(* PLC project BasePpt, Beckhoff Automation GmbH TwinCAT PLC Control 3.5.6.0 *)
(* stored: creationDateTime 2015-05-28T16:00:50.6422414, modificationDateTime 2015-05-28T16:00:50.6452414 *)

TYPE T_Ctrl_SIf_IBH : STRUCT
  Cfg : T_Ctrl_SIf_IBH_Cfg;  (* configuration *)
  Par : T_Ctrl_SIf_IBH_Par;  (* parameter *)
  Cur : T_Ctrl_SIf_IBH_Cur;  (* current values *)
END_STRUCT;
END_TYPE

TYPE T_Ctrl_SIf_IBH_Cfg : STRUCT
  uiNumberOfModules : UINT;  (* Number of Modules in use, <= 8 *)
  tIpAddress : T_IPv4Addr;  (* IPv4 network address *)
  udiPortAdress : UDINT;  (* Remote (server) port address *)
  nDeviceAddress : BYTE;  (* MPI device address *)
  nDatablockNumber : BYTE;  (* Read/write from/to datablock number *)
  tTimeout : TIME;  (* Maximum time allowed for the execution of the command *)
  nWriteStartAddress : WORD;  (* Write byte/word offset/start address *)
  nReadStartAddress : WORD;  (* Read byte/word offset/start address *)
  uiByteOffset_rd_iStatus : UINT;
  uiByteOffset_rd_bOff : UINT;
  uiBitOffset_rd_bOff : UINT;
  uiByteOffset_rd_bBeltOn : UINT;
  uiBitOffset_rd_bBeltOn : UINT;
  uiByteOffset_rd_bManual : UINT;
  uiBitOffset_rd_bManual : UINT;
  uiByteOffset_rd_bRun : UINT;
  uiBitOffset_rd_bRun : UINT;
  uiByteOffset_rd_bSetParam : UINT;
  uiBitOffset_rd_bSetParam : UINT;
  uiByteOffset_rd_bGetParam : UINT;
  uiBitOffset_rd_bGetParam : UINT;
  uiByteOffset_rd_bAckError : UINT;
  uiBitOffset_rd_bAckError : UINT;
  uiByteOffset_rd_adiTemp_mc : UINT;
  uiByteOffset_rd_adiAir_p : UINT;
  uiByteOffset_rd_diSpeed_mm_min : UINT;
  uiByteOffset_rd_iErrorLevel : UINT;
  uiByteOffset_rd_iErrorID : UINT;
  uiByteOffset_rd_iErrorValue : UINT;
  uiByteOffset_wr_iOff : UINT;
  uiByteOffset_wr_iBeltOn : UINT;
  uiByteOffset_wr_iManual : UINT;
  uiByteOffset_wr_iRun : UINT;
  uiByteOffset_wr_iSetParam : UINT;
  uiByteOffset_wr_iGetParam : UINT;
  uiByteOffset_wr_iAckError : UINT;
  uiByteOffset_wr_adiTemp_mc : UINT;
  uiByteOffset_wr_adiAir_p : UINT;
  uiByteOffset_wr_diSpeed_mm_min : UINT;
END_STRUCT;
END_TYPE

TYPE T_Ctrl_SIf_IBH_Cur : STRUCT

END_STRUCT;
END_TYPE

TYPE T_Ctrl_SIf_IBH_Par : STRUCT

END_STRUCT;
END_TYPE

TYPE E_AmpType : (BOTH_ROT_LIN := 0, ROTARY_AMP := 1, LINEAR_AMP := 2) USINT;
END_TYPE

(* values of E_POD_UseHomeSwitch: SI0: internal IO 2 Home switch 0: Switched off, 1: Switched on; SI1: internal IO 16 SI0: 0: Switched off (Open),1: Switched on (Close); SI2: internal IO 17 SI0: 0: Switched off (Open),1: Switched on (Close); SI3: internal IO 18 SI0: 0: Switched off (Open),1: Switched on (Close); SI4: internal IO 19 SI0: 0: Switched off (Open),1: Switched on (Close); SI5: internal IO 20 SI0: 0: Switched off (Open),1: Switched on (Close); SI6: internal IO 21 SI0: 0: Switched off (Open),1: Switched on (Close) internal IO 22 SI0: 0: Switched off (Open),1: Switched on (Close) *)

TYPE E_POD_UseHomeSwitch : (FUB_Input := 0, HomeSwitch, SI0, SI1, SI2, SI3, SI4, SI5, SI6) USINT;
END_TYPE

TYPE E_ValueType : (TYPE_NOT_SPECIFIED := 0, TYPE_SINT := 1, TYPE_INT := 2, TYPE_DINT := 3, TYPE_USINT := 4, TYPE_UINT := 5, TYPE_UDINT := 6, TYPE_STRING := 7) USINT;
END_TYPE

TYPE T_POD : STRUCT
  strAxisName : STRING(31);
  strState : STRING;
  strCmd : STRING;
  intCmd : INT;
  intServiceCmd : INT;
  stStatus : T_POD_Status;
  stMove : T_POD_Move;
  stErr : T_POD_Error;
  stCfg : T_POD_Cfg;
  stService : T_POD_Service;
END_STRUCT;
END_TYPE

TYPE T_POD_Cfg : STRUCT
  bolSimulation : BOOL;
  lreHomePosition : LREAL;  (* >0 Homeposition set if calibsignal active *)
  eHomingMode : MC_HomingMode;  (* Home Mode *)
  eUseHomeSwitch : E_POD_UseHomeSwitch;  (* define home switch: 0 use FUB input, *)
END_STRUCT;
END_TYPE

TYPE T_POD_DigitalInputs : STRUCT
  bol_N_OT : BOOL;  (* 0 N-OT: Negative limit switch 0: Switched off, 1: Switched on *)
  bol_P_OT : BOOL;  (* 1 P-OT: Positive limit switch 0: Switched off, 1: Switched on *)
  bol_HomeSwitch : BOOL;  (* 2 Home switch 0: Switched off, 1: Switched on *)
  bol_SI0 : BOOL;  (* 16 SI0: CN1-13pin 0: Switched off (Open),1: Switched on (Close) *)
  bol_SI1 : BOOL;  (* 17 SI1: CN1-7pin 0: Switched off (Open),1: Switched on (Close) *)
  bol_SI2 : BOOL;  (* 18 SI2: CN1-8pin 0: Switched off (Open),1: Switched on (Close) *)
  bol_SI3 : BOOL;  (* 19 SI3: CN1-9pin 0: Switched off (Open),1: Switched on (Close) *)
  bol_SI4 : BOOL;  (* 20 SI4: CN1-10pin 0: Switched off (Open),1: Switched on (Close) *)
  bol_SI5 : BOOL;  (* 21 SI5: CN1-11pin 0: Switched off (Open),1: Switched on (Close) *)
  bol_SI6 : BOOL;  (* 22 SI6: CN1-12pin 0: Switched off (Open),1: Switched on (Close) *)
END_STRUCT;
END_TYPE

TYPE T_POD_Error : STRUCT
  bolErrAck : BOOL;  (* Reset failure *)
  bolErrorActive : BOOL;  (* atleast one failure active *)
  bolMCError : BOOL;  (* error in MC fub error *)
  bolNCError : BOOL;  (* error in NC (motion controller) *)
  bolDriveError : BOOL;  (* error in drive (ELMO) *)
  dwoErrorID : DWORD;  (* error ID *)
END_STRUCT;
END_TYPE

TYPE T_POD_Move : STRUCT
  lreSetPos : LREAL;  (* target position [Units] *)
  eDirection : MC_Direction;  (* Direction used for Modulo position *)
  lreSetSpeed : LREAL;  (* set speed [Units/s] *)
  lreSetAcc : LREAL;  (* set acc [Units/s^2] *)
  lreSetDec : LREAL;  (* set dec [Units/s^2] *)
  lreSetDecFast : LREAL;  (* set dec [Units/s^2] quickstop *)
  lreSetJerk : LREAL;  (* lreSetDec : DINT; //set dec [Units/s^2] *)
  lreSpeedOverride : LREAL := 100.0;  (* speed override for all drive commands (0 ≤Override≤ 100.0) *)
  lreSWLimitNeg_mm : LREAL;
  lreSWLimitPos_mm : LREAL;
  lreActPos : LREAL;  (* Actual position [Units] *)
  lreActModPos : LREAL;  (* Actual modulo position [Units] *)
  lreActVel : LREAL;  (* act speed [Units/s] *)
  lreActTorque : LREAL;  (* [Nm] actual torque The torque actual value corresponds to the instantaneous torque in the drive motor. The value is given in units of per thousand of rated torque. *)
END_STRUCT;
END_TYPE

TYPE T_POD_Service : STRUCT
  worIndex : WORD;  (* Index of the object that should be written to. *)
  bytSubIndex : BYTE;  (* Sub-index of the object that should be written to. *)
  dwo_pSrcBuf : DWORD;  (* Address (pointer) of the send buffer. *)
  udi_cbBufLen : UDINT;  (* Number (in bytes) of data to be sent. *)
  eValueType : E_ValueType;  (* value type *)
  eNC_ParNumber : MC_AxisParameter;  (* parameter number of read/write NC parameters *)
  strValue : STRING;  (* write/read value if dwo_pSrcBuf = 0 *)
END_STRUCT;
END_TYPE

TYPE T_POD_StateMachine : STRUCT
  intState : INT;  (* actual state *)
  intStateLastCycle : INT;  (* state of last cycle *)
  intStateHistory : INT;  (* save history backup p.e. in ERROR state *)
  intStateNext : INT;  (* set state for next cycle *)
END_STRUCT;
END_TYPE

TYPE T_POD_Status : STRUCT
  bolEnable : BOOL;  (* Hardware enable:0 = Open 1 = Closed *)
  bolNetwOk : BOOL;  (* 1 = Network initialized *)
  bolInitOk : BOOL;  (* 1 = Initialization done *)
  bolReady : BOOL;
  bolCtrlOn : BOOL;  (* 1 = Controller switched on *)
  bolHomeOk : BOOL;  (* 1 = Homing done *)
  bolInPos : BOOL;  (* 1 = In position (target position reached) *)
  bolMoving : BOOL;  (* 1 = Axis moving *)
  bolNegHWSwitch : BOOL;  (* 1 = negativ endswitch active -> no movement negative allowed *)
  bolPosHWSwitch : BOOL;  (* 1 = positive endswitch active -> no movement positive allowed *)
  bolNegSWSwitch : BOOL;  (* 1 = negativ endswitch active -> no movement negative allowed *)
  bolPosSWSwitch : BOOL;  (* 1 = positive endswitch active -> no movement positive allowed *)
  stDigIn : T_POD_DigitalInputs;  (* drive digital inputs of elmo drive *)
END_STRUCT;
END_TYPE

TYPE T_POD_StatusWord : STRUCT
  bolReadyToSwitchOn : BOOL;  (* 0 Ready TO Switch on =1 *)
  bolSwitchedOn : BOOL;  (* 1 Switched on =1 *)
  bolOperationEnabled : BOOL;  (* 2 Operation enabeld =1 *)
  bolFault : BOOL;  (* 3 Fault/Fault Reaction *)
  bolMainPowerOn : BOOL;  (* 4 MainPower on =1 *)
  bolQuickStopInactive : BOOL;  (* 5 Quickstop inaktive =1 *)
  bolSwitchOnDisabled : BOOL;  (* 6 Switch on disabled =1 *)
  bolWarning : BOOL;  (* 7 Warning is occurred =1 *)
  bolBit08 : BOOL;  (* 8 not used always 0 *)
  bolRemote : BOOL;  (* 9 The Remote bit is always set by the Elmo servo drive *)
  bolTargetReached : BOOL;  (* 10 Target Reached *)
  bolInternLimit : BOOL;  (* 11 Internal Limit active =1 *)
END_STRUCT;
END_TYPE

TYPE E_PTR_Status : (EnterBusy, OnBelt, ExitBusy, Gone, ERROR, MAX_E_PTR_Status);
END_TYPE

TYPE T_PTR_STRUCT : STRUCT
  udiTimeOnBelt_us : UDINT;  (* [us] Time of the paper on the belt *)
  lrePositionOnBelt_mm : LREAL;  (* [mm] Position of the paper on the belt *)
  lrePositionOnBeltAdjusted_mm : LREAL;  (* [mm] Position of the paper on the belt Adjusted to the possible maximum *)
  udiItemId : UDINT;  (* Paper Item Id *)
  eStatus : E_PTR_Status;  (* Error *)
END_STRUCT;
END_TYPE

TYPE E_ALM_TCP : (SocketConnectionLost := 1, AddToSendBufferFailed := 2, RemoveFromSendBufferFailed := 3, GetFromSendBufferFailed := 4, AddToReceiveBufferFailed := 5, RemoveFromReceiveBufferFailed := 6, GetFromReceiveBufferFailed := 7, NotSent := 8, NoAckReceived := 9, FubErrorClientConnection := 10, FubErrorSendData := 11, FubErrorReceiveData := 12, MAX_E_ALM_TCP) UINT;
END_TYPE

{attribute 'pack_mode' := '1'}
TYPE ST_Header : STRUCT
  uinMsgId : UINT;
  udiMsgSize : UDINT;
END_STRUCT;
END_TYPE

TYPE T_Ctrl_SIf_TCP : STRUCT
  Cfg : T_Ctrl_SIf_TCP_Cfg;  (* configuration *)
  Par : T_Ctrl_SIf_TCP_Par;  (* parameter *)
  Cur : T_Ctrl_SIf_TCP_Cur;  (* current values *)
  Alm : ARRAY[1..(E_ALM_TCP.MAX_E_ALM_TCP - 1)] OF T_Ctrl_Alm;  (* alarm number used in this controller *)
END_STRUCT;
END_TYPE

TYPE T_Ctrl_SIf_TCP_Cfg : STRUCT
  bUsingAck : BOOL;  (* depending on the protocol an ACK is used or not *)
  bolAutoReconnectEnable : BOOL;  (* Enable Auto Reconnect *)
END_STRUCT;
END_TYPE

TYPE T_Ctrl_SIf_TCP_Cur : STRUCT
  bolFubErrorActive : BOOL;
END_STRUCT;
END_TYPE

TYPE T_Ctrl_SIf_TCP_Par : STRUCT
  strIPAdr : STRING(15);
  udiPort : UDINT;
  tTOConnection : TIME;
  tTOReceive : TIME;
  tTOSend : TIME;
  iMaxWaitTimeAck : TIME;
  iMaxSendTry : USINT;
END_STRUCT;
END_TYPE

TYPE E_ALM_GRR : (NONE := 1, SystemError := 2, MainPressureError := 3, EoffOrFuseError := 4, LowPowderWarning := 5, ManualOperation := 6, LostConnection := 7, MAX_E_ALM_GRR) UINT;
END_TYPE

TYPE T_Ctrl_SIf_GRR : STRUCT
  Cfg : T_Ctrl_SIf_GRR_Cfg;  (* configuration *)
  Par : T_Ctrl_SIf_GRR_Par;  (* parameter *)
  Cur : T_Ctrl_SIf_GRR_Cur;  (* current values *)
  In : T_Ctrl_SIf_GRR_In;  (* io input *)
  Out : T_Ctrl_SIf_GRR_Out;  (* io output *)
  Alm : ARRAY[1..(E_ALM_GRR.MAX_E_ALM_GRR - 1)] OF T_Ctrl_Alm;  (* alarm number used in this controller *)
END_STRUCT;
END_TYPE

TYPE T_Ctrl_SIf_GRR_Cfg : STRUCT
  rMaxFreq_Hz : REAL;
END_STRUCT;
END_TYPE

TYPE T_Ctrl_SIf_GRR_Cur : STRUCT
  intMainPressure : INT;
END_STRUCT;
END_TYPE

TYPE T_Ctrl_SIf_GRR_In : STRUCT
  bolSystemOk : T_Ctrl_IoBool;
  bolMainPressureError : T_Ctrl_IoBool;
  bolEoffOrFuseOk : T_Ctrl_IoBool;
  bolPowderLowWarning : T_Ctrl_IoBool;
  bolAutoMode : T_Ctrl_IoBool;
  intState : T_Ctrl_IoInt;
  bolToggleBitGrn : T_Ctrl_IoBool;
  intMainPressure : T_Ctrl_IoInt;
END_STRUCT;
END_TYPE

TYPE T_Ctrl_SIf_GRR_Out : STRUCT
  intCommand : BASE_PLC.T_Ctrl_IoInt;
  intConveyorBelt : T_Ctrl_IoInt;
  intPowderVibrator : T_Ctrl_IoInt;
  intConveyorVibrator : T_Ctrl_IoInt;
  intAnalogValue : T_Ctrl_IoInt;
  uinFilterClearingCycleTime_min : T_Ctrl_IoUint;
  bolToggleBitGrr : T_Ctrl_IoBool;
END_STRUCT;
END_TYPE

TYPE T_Ctrl_SIf_GRR_Par : STRUCT
  rConveyorBelt_Hz : REAL;
  rPowderVibrator_Hz : REAL;
  rConveyorVibrator_Hz : REAL;
  rAnalogValue_p : REAL;
  uinFilterClearingCycleTime_min : UINT;
END_STRUCT;
END_TYPE

TYPE E_ALM_JCL : (NONE := 1, JetterNotRun := 2, JetterManualWarning := 3, JetterManualError := 4, JetterEOff := 5, JetterCommunicationLost := 6, CleaningError, MAX_E_ALM_JCL) UINT;
END_TYPE

TYPE T_Ctrl_SIf_JCL : STRUCT
  Cfg : T_Ctrl_SIf_JCL_Cfg;  (* configuration *)
  Par : T_Ctrl_SIf_JCL_Par;  (* parameter *)
  Cur : T_Ctrl_SIf_JCL_Cur;  (* current values *)
  Alm : ARRAY[1..(E_ALM_JCL.MAX_E_ALM_JCL - 1)] OF T_Ctrl_Alm;  (* alarm number used in this controller *)
END_STRUCT;
END_TYPE

TYPE T_Ctrl_SIf_JCL_Cfg : STRUCT
  bolJetterManualModeAllowed : BOOL;  (* FALSE = Do not allow manual mode, go to error if Jetter goes to manual / TRUE = Allow manual mode and stay in the last state *)
END_STRUCT;
END_TYPE

TYPE T_Ctrl_SIf_JCL_Cur : STRUCT
  bolIsLocalControlled : BOOL;  (* Additional states from TCP server Local control active. Commands from this client are ignored *)
  bolIsRemoteControlled : BOOL;  (* Remote control active. Commands from this client are accepted *)
  bolReadyForProduction : BOOL;  (* Jetter ready for production *)
  bolMaintenanceInProgress : BOOL;  (* TRUE if a maintenance work is in progress. Independent if auto or manual maintenance is in progress. *)
  bolRunning : BOOL;  (* Print running, in production *)
  bolNeedsAttention : BOOL;  (* System needs attention. Info or warning active *)
  bolError : BOOL;  (* General error active *)
  bolCleaningIncomplete : BOOL;  (* Cleaning cycle was aborted before finishing. Production not possible. *)
  bolNeedsCleaning : BOOL;  (* Print head needs cleaning. *)
  strDTOfLastCleaningCycle : STRING := '';  (* Timestamp of the last cleaning cycle. Format: YYYY-MM-DD-hh:mm:ss.xxx *)
  intJETState : INT;  (* Jetter state *)
END_STRUCT;
END_TYPE

TYPE T_Ctrl_SIf_JCL_Par : STRUCT
  udiCleaningStartTimeout_ms : UDINT;  (* [ms] Timeout to detect cleaning start failure *)
END_STRUCT;
END_TYPE

TYPE T_JCL_AlmMsg : STRUCT
  stHeader : ST_Header;
  udiAlarmID : UDINT;  (* Unique alarm number *)
  udiInfo : UDINT;  (* Additional information *)
  usiClass : USINT;  (* Corresponding alarm class *)
  uinCtrlID : UINT;  (* Corresponding controller ID *)
  strDTEntry : STRING(25);  (* Entry date and time *)
  strText : STRING(255);  (* Alarm Text *)
END_STRUCT;
END_TYPE

{attribute 'pack_mode' := '1'}
TYPE T_JCL_Command : STRUCT
  stHeader : ST_Header;
  usiCommand : USINT;
END_STRUCT;
END_TYPE

TYPE T_JCL_PrintDone : STRUCT
  stHeader : ST_Header;
  usiBarcode : ARRAY[0..9] OF USINT;
  usiInkLevelMainTank : USINT;  (* [%] *)
  usiInkLevelSupplyPrintModule1 : USINT;  (* [%] *)
  usiInkLevelSupplyPrintModule2 : USINT;  (* [%] *)
  usiInkLevelReturnPrintModule1 : USINT;  (* [%] *)
  usiInkLevelReturnPrintModule2 : USINT;  (* [%] *)
  udiInkMeniscus : ARRAY[0..1] OF UDINT;  (* [0.01 mbar] *)
  udiPrintHeadTemperature : ARRAY[0..1, 0..4] OF UDINT;  (* [0.1 °C] *)
  udiPrintWidthCalc : UDINT;  (* [Micrometer] // Dimension of printed file calculated by DJM *)
  udiPrintLengthCalc : UDINT;  (* [Micrometer] // Dimension of printed file calculated by DJM *)
  udiShiftXCalc : UDINT;  (* [Micrometer] // Offset of print *)
  udiShiftYCalc : UDINT;  (* [Micrometer] // Offset of print *)
  udiShiftAngleCalc : UDINT;  (* [0.01°] // Offset of rotation angle *)
END_STRUCT;
END_TYPE

{attribute 'pack_mode' := '1'}
TYPE T_JCL_RequestCleaning : STRUCT
  stHeader : ST_Header;
  strDTLastClean : STRING(25);  (* Date and time of the last cleaning cycle *)
  uinRequiredInterval_min : UINT;  (* Required interval for cleaning [min] *)
END_STRUCT;
END_TYPE

{attribute 'pack_mode' := '1'}
TYPE T_JCL_State : STRUCT
  stHeader : ST_Header;
  usiMainState : USINT;
  usiAddState : USINT;  (* (Bit coded) *)
END_STRUCT;
END_TYPE

{attribute 'qualified_only'}
TYPE E_ALM_RAX : (GeneralDrive := 1, GeneralNc, SwLimit, NegHwLimit, PosHwLimit, InterlockNegMove, InterlockPosMove, GeneralMCFUB, MAX_E_ALM) UINT;
END_TYPE

TYPE T_Ctrl_SIf_RAX : STRUCT
  Cfg : T_Ctrl_SIf_RAX_Cfg;  (* configuration *)
  Par : T_Ctrl_SIf_RAX_Par;  (* parameter *)
  Cur : T_Ctrl_SIf_RAX_Cur;  (* current values *)
  Alm : ARRAY[1..(E_ALM_RAX.MAX_E_ALM - 1)] OF T_Ctrl_Alm;  (* alarm number used in this controller *)
  Ilk : T_Ctrl_SIf_RAX_Ilk;  (* interlock of output/movements *)
END_STRUCT;
END_TYPE

TYPE T_Ctrl_SIf_RAX_Cfg : STRUCT
  eHomingMode : MC_HomingMode;  (* homing mode *)
  lreShortestWayWindow_deg : LREAL;
END_STRUCT;
END_TYPE

TYPE T_Ctrl_SIf_RAX_Cur : STRUCT
  dinSpeed_0_1deg_s : DINT;  (* [0.1°/s] current speed *)
  dinPosition_0_1deg : DINT;  (* [0.1°] current position *)
  dinModPosition_0_1deg : DINT;  (* [°] current modulo position *)
  dinTorque_0_1Nm : DINT;  (* [0.1Nm] current torque *)
  bol_di1 : BOOL;  (* digital input1 from drive *)
  bol_di2 : BOOL;  (* digital input2 from drive *)
  bol_di3 : BOOL;  (* digital input3 from drive *)
  bol_di4 : BOOL;  (* digital input4 from drive *)
  bol_di5 : BOOL;  (* digital input5 from drive *)
END_STRUCT;
END_TYPE

TYPE T_Ctrl_SIf_RAX_Ilk : STRUCT
  bolMovePos : BOOL;  (* interlock movment in positive direction *)
  bolMoveNeg : BOOL;  (* interlock movment in negative direction *)
END_STRUCT;
END_TYPE

TYPE T_Ctrl_SIf_RAX_Par : STRUCT
  dinHomeOffset_0_1deg : DINT;  (* [deg] home offset *)
  dinPositionInit_0_1deg : DINT;  (* [0.1°] position init *)
  dinPos_0_1deg : DINT;  (* [0.1°] position absolute *)
  dinRelDist_0_1deg : DINT;  (* [0.1°] rel distance *)
  dinSpeed_0_1deg_s : DINT;  (* [0.1°/s] position speed *)
  dinSpeed_per : DINT;  (* [%] percent from dinSetSpeed_0_1deg_s *)
  dintAccDec_0_1deg_s2 : DINT;  (* [0.1°/s^2] position acceleration *)
  dinAcc_per : DINT;  (* [%] percent from dintAccDec_0_1deg_s2 *)
  dinDec_per : DINT;  (* [%] percent from dintAccDec_0_1deg_s2 *)
  dinSetDecFast_0_1deg_s2 : DINT;  (* [0.1°/s^2] position deceleration fast em stop *)
  dinSWLimitNeg_0_1deg : DINT;  (* [0.1°] negative sw limite *)
  dinSWLimitPos_0_1deg : DINT;  (* [0.1°] positive sw limite *)
END_STRUCT;
END_TYPE

TYPE E_ALM_BCH : (DataChannelMissing := 1, DataChannelBufferFull, BarcodeNotReadCorrectly, MAX_E_ALM_BCH) UINT;
END_TYPE

TYPE T_Ctrl_SIf_BCH : STRUCT
  Cfg : T_Ctrl_SIf_BCH_Cfg;  (* configuration *)
  Par : T_Ctrl_SIf_BCH_Par;  (* parameter *)
  Cur : T_Ctrl_SIf_BCH_Cur;  (* current values *)
  In : T_Ctrl_SIf_BCH_In;  (* Input layer *)
  Alm : ARRAY[1..(E_ALM_BCH.MAX_E_ALM_BCH - 1)] OF T_Ctrl_Alm;  (* alarm number used in this controller *)
END_STRUCT;
END_TYPE

TYPE T_Ctrl_SIf_BCH_Cfg : STRUCT
  bolEnableDataChannel : BOOL;  (* TRUE = Enable Data Channel; False = Disable DataChannel *)
  bolNegativeTriggerSignal : BOOL;  (* TRUE = Negative Trigger Signal, FALSE = Positive Trigger Signal *)
END_STRUCT;
END_TYPE

TYPE T_Ctrl_SIf_BCH_Cur : STRUCT

END_STRUCT;
END_TYPE

TYPE T_Ctrl_SIf_BCH_In : STRUCT
  bolSensorTrigScan : BASE_PLC.T_Ctrl_IoBool;  (* Trigger the measurement sensor *)
END_STRUCT;
END_TYPE

TYPE T_Ctrl_SIf_BCH_Par : STRUCT
  udiPaperGoneDelay_ms : UDINT;  (* [ms] Delay after the barcode has be read and the paper sensor signals that the paper is gone *)
  udiTestReadCylceTime_ms : UDINT;  (* [ms] Test Read Cycle Time *)
END_STRUCT;
END_TYPE

TYPE E_ALM_MDC : (TableSensorTimeout := 1, CrossSensorTimeout := 2, PositionSame := 3, MAX_E_ALM_MDC);
END_TYPE

TYPE T_Ctrl_SIf_MDC : STRUCT
  Cfg : T_Ctrl_SIf_MDC_Cfg;  (* configuration *)
  Par : T_Ctrl_SIf_MDC_Par;  (* parameter *)
  Cur : T_Ctrl_SIf_MDC_Cur;  (* current values *)
  In : T_Ctrl_SIf_MDC_In;  (* io input *)
  Out : T_Ctrl_SIf_MDC_Out;  (* io output *)
  Alm : ARRAY[1..MAX_E_ALM_MDC] OF T_Ctrl_Alm;  (* alarm number used in this controller *)
  Ilk : T_Ctrl_SIf_MDC_Ilk;  (* interlock of output/movements *)
END_STRUCT;
END_TYPE

TYPE T_Ctrl_SIf_MDC_Cfg : STRUCT
  uintPositionPerTurn : UINT;  (* Number of positions in 360° of the Malteser drive *)
END_STRUCT;
END_TYPE

TYPE T_Ctrl_SIf_MDC_Cur : STRUCT
  uintActualPosition : UINT;  (* Actual Position as position *)
  eActualTurningDirection : E_TURN_DIRECTION;  (* actual turning direction *)
  bolReferenceOk : BOOL;  (* Reference still ok *)
END_STRUCT;
END_TYPE

TYPE T_Ctrl_SIf_MDC_Ilk : STRUCT

END_STRUCT;
END_TYPE

TYPE T_Ctrl_SIf_MDC_In : STRUCT
  bolCrossPositionSensor : BASE_PLC.T_Ctrl_IoBool;  (* Is the cross in sensor positinon. One rotation step done. *)
  bolTablePositionSensor : BASE_PLC.T_Ctrl_IoBool;  (* Is the table at 0° degrees *)
END_STRUCT;
END_TYPE

TYPE T_Ctrl_SIf_MDC_Out : STRUCT
  intActualPosition : BASE_PLC.T_Ctrl_IoInt;
END_STRUCT;
END_TYPE

TYPE T_Ctrl_SIf_MDC_Par : STRUCT
  intTurnDirection : INT;  (* <0 = Turn left; =0 automatic; >0 turn right *)
  uinPositionToGo : UINT;  (* Position to go to if comand turn is given. 0 = initialization position *)
  udiStepRotationTime_ms : UDINT;  (* [ms] time to rotate one step *)
  udiInitializationTime_ms : UDINT;  (* [ms] initialization timeout time *)
  udiSimStepRotationTime_ms : UDINT;  (* [ms] simulation time to rotate one step *)
  udiSimInitializationTime_ms : UDINT;  (* [ms] simulation initialization timeout time *)
  udiSimStartRotationTime_ms : UDINT;  (* [ms] simulation time to start rotate and Cross sensor needs to go away *)
  uinPrePositionSpeed_rpm : UINT;  (* [rpm] PrePosition Speed *)
  uinPositionSpeed_rpm : UINT;  (* [rpm] Position Speed *)
END_STRUCT;
END_TYPE

(* values of E_ALM_OVN: Tesoma10000: OvertemperaturePowerSection - software reset - operating mode must be reelected; Tesoma10002: FailureOfActiveCoolingUnit; Tesoma10003: ActiveCoolingUnitNotRunning; Tesoma10006: FailureFuseGeneral - transport starts immediately when sensor is free; Tesoma10010: BeltPositionControlSensorError - software reset; Tesoma10011: BeltEdgeShutOff - software reset; Tesoma10012: FaultBeltSpeed - software reset; Tesoma10013: TransportOverload; Tesoma10014: BeltControlDeviceFault - software reset - reset FC; Tesoma10016: EmergencyStop - would be resettable, but since power is gone, the acknowledge does not arrive; Tesoma10023: BeltWearMonitor; Tesoma10024: ControlCabinetFan; Tesoma10025: ControlCabinetTemperatureTooHigh; Tesoma10026: PowerSupplyFailure; Tesoma10027: IntakeHoodTemperatureExceeded; Tesoma10030: AirPressureTooLow; Tesoma10031: BeltPositionControlNotWorking; Tesoma10032: ErrorCoolingDeviceControlCabinet; Tesoma10034: ControlCabinetCoolerAndSmallDrivesFuseFailure; Tesoma10x00: LimitSwitchingOff - software reset - after elimination, reactivates according zone; Tesoma10x01: OvertemperatureStl - software reset - after elimination AND reset, the STL reactivates the accordant zone; Tesoma10x02: FuseTriggered - software reset - after elimination, reactivates the accordant zone; Tesoma10x03: FailureExhaustAirDps - software reset - after elimination, reactivates the accordant zone; Tesoma10x07: ErrorFrequencyConverter - software reset - after elimination AND reset, the FC reactivates the accordant zone; Tesoma10x13: TemperatureSensorIrDefective; Tesoma10x14: FaultFrameCoolingSystemDps; Tesoma10x15: FaultExhaustAirDps; Tesoma13x00: TemperatureFault - software reset *)

TYPE E_ALM_OVN : (NONE := 0, TempError := 1, AirError := 2, SpeedError := 3, TimeoutError := 4, ParameterWarning := 5, ConnectionError := 6, WrongMode := 7, Tesoma10000 := 8, Tesoma10002 := 9, Tesoma10003 := 10, Tesoma10006 := 11, Tesoma10010 := 12, Tesoma10011 := 13, Tesoma10012 := 14, Tesoma10013 := 15, Tesoma10014 := 16, Tesoma10016 := 17, Tesoma10023 := 18, Tesoma10024 := 19, Tesoma10025 := 20, Tesoma10026 := 21, Tesoma10027 := 22, Tesoma10030 := 23, Tesoma10031 := 24, Tesoma10032 := 25, Tesoma10034 := 26, Tesoma10x00 := 27, Tesoma10x01 := 28, Tesoma10x02 := 29, Tesoma10x03 := 30, Tesoma10x07 := 31, Tesoma10x13 := 32, Tesoma10x14 := 33, Tesoma10x15 := 34, Tesoma13x00 := 35, TesomaUnknown := 36, HostConnectionLost := 37, SettingsChanged := 38, MAX_E_ALM_OVN);
END_TYPE

TYPE T_Ctrl_SIf_OVN : STRUCT
  Cfg : T_Ctrl_SIf_OVN_Cfg;  (* configuration *)
  Par : T_Ctrl_SIf_OVN_Par;  (* parameter *)
  Cur : T_Ctrl_SIf_OVN_Cur;  (* current values *)
  In : T_Ctrl_SIf_OVN_In;  (* io input *)
  Out : T_Ctrl_SIf_OVN_Out;  (* io output *)
  Alm : ARRAY[1..(E_ALM_OVN.MAX_E_ALM_OVN - 1)] OF T_Ctrl_Alm;  (* alarm number used in this controller *)
END_STRUCT;
END_TYPE

TYPE T_Ctrl_SIf_OVN_Cfg : STRUCT
  uiNumberOfModules : UINT;  (* Number of Modules in use *)
  diModuleLength_mm : DINT;  (* Length of one Module *)
  diDistanceBeforeOven_mm : DINT;  (* Distance before the first Module *)
  diDistanceAfterOven_mm : DINT;  (* Distance after the last Module *)
  diMaxSpeed_mm_min : DINT;  (* Maximal Belt Speed in mm/min *)
  diMinSpeed_mm_min : DINT;  (* Minimal Belt Speed in mm/min *)
  diMinTemp_dc : DINT;  (* Minimal Temperature in deci °C *)
  diMaxTemp_dc : DINT;  (* Maximal Temperature in deci °C *)
  diMinAir_p : DINT;  (* Minimal Airflow in % *)
  diMaxAir_p : DINT;  (* Maximal Airflow in % *)
  bAutoContinueAfterConnectionError : BOOL;  (* Auto Continue After Connection Error *)
  bolDataChannelEnable : BOOL;  (* Enable Data Channel *)
  bIgnoreOffBusyWaitPaper : BOOL;  (* ignore waiting for Paper to eject in OFFBusy *)
END_STRUCT;
END_TYPE

TYPE T_Ctrl_SIf_OVN_Cur : STRUCT
  diSpeed_mm_min : DINT;  (* Belt Speed in mm/min *)
  adiTemp_dc : ARRAY[0..(MAX_NUMBER_OF_OVEN_MODULES - 1)] OF DINT;  (* Temperature in deci °C *)
  adiAir_p : ARRAY[0..(MAX_NUMBER_OF_OVEN_MODULES - 1)] OF DINT;  (* Airflow in % *)
END_STRUCT;
END_TYPE

TYPE T_Ctrl_SIf_OVN_In : STRUCT

END_STRUCT;
END_TYPE

TYPE T_Ctrl_SIf_OVN_Out : STRUCT

END_STRUCT;
END_TYPE

TYPE T_Ctrl_SIf_OVN_Par : STRUCT
  diSpeed_mm_min : DINT;  (* Belt Speed in mm/min *)
  diSpeedBand1_mm_min : DINT;  (* Belt Speed Band in mm/min *)
  diSpeedBand2_mm_min : DINT;  (* Belt Speed Band in mm/min *)
  udiSpeedTimeout_ms : UDINT;  (* Belt Speed Timeout in ms *)
  adiTemp_dc : ARRAY[0..(MAX_NUMBER_OF_OVEN_MODULES - 1)] OF DINT;  (* Temperature in deci °C *)
  adiTempBand1_dc : ARRAY[0..(MAX_NUMBER_OF_OVEN_MODULES - 1)] OF DINT;  (* Temperature Band in deci °C *)
  adiTempBand2_dc : ARRAY[0..(MAX_NUMBER_OF_OVEN_MODULES - 1)] OF DINT;  (* Temperature Band in deci °C *)
  audiTempTimeout_ms : ARRAY[0..(MAX_NUMBER_OF_OVEN_MODULES - 1)] OF UDINT;  (* Temperature Timeout in ms *)
  adiAir_p : ARRAY[0..(MAX_NUMBER_OF_OVEN_MODULES - 1)] OF DINT;  (* Airflow in % *)
  adiAirBand1_p : ARRAY[0..(MAX_NUMBER_OF_OVEN_MODULES - 1)] OF DINT;  (* Airflow Band in % *)
  adiAirBand2_p : ARRAY[0..(MAX_NUMBER_OF_OVEN_MODULES - 1)] OF DINT;  (* Airflow Band in % *)
  audiAirTimeout_ms : ARRAY[0..(MAX_NUMBER_OF_OVEN_MODULES - 1)] OF UDINT;  (* Airflow Timeout in ms *)
  udiTimeoutOffBusy_ms : UDINT;
  udiTimeoutRunBusyReaction_ms : UDINT;
  udiTimeoutRunBusyInBand_ms : UDINT;
  udiTimeoutBeltOnlyReaction_ms : UDINT;
  udiTimeoutBeltOnlyBusy_ms : UDINT;
END_STRUCT;
END_TYPE

{attribute 'enable_dynamic_creation'}
TYPE T_Data : STRUCT
  uliBarcode : ULINT;
  bTrash : BOOL;
  diDistance_um : DINT;
  diSumTemp_mc : ARRAY[0..(MAX_NUMBER_OF_OVEN_MODULES - 1)] OF DINT;
  diCyclesInModule : ARRAY[0..(MAX_NUMBER_OF_OVEN_MODULES - 1)] OF DINT;
  bBarcodeMissed : BOOL;
END_STRUCT;
END_TYPE

TYPE E_ALM_PTB : (TestAlarm := 1, MAX_E_ALM_PTB);
END_TYPE

TYPE E_BELT_DIRECTION : (FORWARD := 0, BACKWARD := 1, MAX_E_BELT_DIRECTION);
END_TYPE

(* values of E_PTB_MODE: Endless: 0; ToSensor: 1; ToDistance: 2; ToTime: 3; Stack: 4 *)

TYPE E_PTB_MODE : (Endless, ToSensor, ToDistance, ToTime, Stack, MAX_E_PTB_MODE);
END_TYPE

TYPE E_PTB_PaperDirection : (Portrait, Landscape, MAX_E_PTB_PaperDirection);
END_TYPE

TYPE T_Ctrl_SIf_PTB : STRUCT
  Cfg : T_Ctrl_SIf_PTB_Cfg;  (* configuration *)
  Par : T_Ctrl_SIf_PTB_Par;  (* parameter *)
  Cur : T_Ctrl_SIf_PTB_Cur;  (* current values *)
  In : T_Ctrl_SIf_PTB_In;  (* io input *)
  Out : T_Ctrl_SIf_PTB_Out;  (* io output *)
  Alm : ARRAY[1..E_ALM_PTB.MAX_E_ALM_PTB] OF T_Ctrl_Alm;  (* alarm number used in this controller *)
  Ilk : T_Ctrl_SIf_PTB_Ilk;  (* interlock of output/movements *)
END_STRUCT;
END_TYPE

TYPE T_Ctrl_SIf_PTB_Cfg : STRUCT
  eMode : E_PTB_MODE;  (* Function Mode *)
  bolVacuumPresent : BOOL;  (* Vacuum pump present *)
  udiBeltLength_mm : UDINT;  (* [mm] Length of the belt *)
  rBeltParam : T_Belt_Cfg_Base;  (* Belt Parameter *)
  bolEntrySensorDebounceEnable : BOOL;  (* Enable Entry Belt Sensor Debounce *)
  bolExitSensorDebounceEnable : BOOL;  (* Enable Exit Belt Sensor Debounce *)
END_STRUCT;
END_TYPE

TYPE T_Ctrl_SIf_PTB_Cur : STRUCT
  eActualDirection : E_BELT_DIRECTION;  (* actual belt direction *)
  udiDistanceToMove_mm : UDINT;  (* [mm] Distance to move if Move Mode is distance *)
  udiTimeToMove_ms : UDINT;  (* [ms] Time to move *)
  rBeltParam : T_Belt_Cur_Base;  (* Belt parameter *)
  udiBeltTimeBase_mm : UDINT;  (* Belt Run Time *)
  uinPaperOnBelt : UINT;  (* Paper on the belt *)
  pPositionList : POINTER TO T_PTR_STRUCT;  (* Pointer to the Position list of the paper on the belt *)
END_STRUCT;
END_TYPE

TYPE T_Ctrl_SIf_PTB_Ilk : STRUCT

END_STRUCT;
END_TYPE

TYPE T_Ctrl_SIf_PTB_In : STRUCT
  bolBeltEntrySensor : BASE_PLC.T_Ctrl_IoBool;
  bolBeltExitSensor : BASE_PLC.T_Ctrl_IoBool;
  bolBeltEntrySensorPEdge : BASE_PLC.T_Ctrl_IoBool;
  bolBeltEntrySensorNEdge : BASE_PLC.T_Ctrl_IoBool;
  bolBeltExitSensorPEdge : BASE_PLC.T_Ctrl_IoBool;
  bolBeltExitSensorNEdge : BASE_PLC.T_Ctrl_IoBool;
END_STRUCT;
END_TYPE

TYPE T_Ctrl_SIf_PTB_Out : STRUCT

END_STRUCT;
END_TYPE

TYPE T_Ctrl_SIf_PTB_Par : STRUCT
  intDirection : INT;  (* <0 = Backward; =0 None; >0 forward *)
  udiDistanceToMove_mm : UDINT;  (* [mm] Distance to move if Move Mode is distance *)
  udiTimeToMove_ms : UDINT;  (* [ms] Time to move *)
  uinPaperStackHight : UINT;  (* Stack hight in # of sheets *)
  bolAutoEjectAfterStack : BOOL;  (* Automatic ejecting the paper if stackhight is reached *)
  bolAutoStackAfterEject : BOOL;  (* Automatic stacking the paper after ejecting all paper *)
  rBeltParam : T_Belt_Par_Base;  (* Belt Parameter *)
  udiStackDelayTime_ms : UDINT;  (* [ms] Stack delay time - Delay before out motor can move after paper entered system *)
  udiBeltLength_mm : UDINT;  (* [mm] Belt Length *)
  ePaperOrientation : E_PTB_PaperDirection;  (* Page running format *)
  uinPaperHight_mm : UINT;  (* [mm] Paper Hight *)
  uinPaperWidth_mm : UINT;  (* [mm] Paper Width *)
  uinInputSignalDebounceTime_ms : UINT;  (* [ms] Input Parameter Debounce time *)
END_STRUCT;
END_TYPE

TYPE E_ALM_PBC : (PaperTransport := 1, BufferFull := 2, BufferEmpty := 3, DoublePaperError := 4, DataChannelBufferFull := 5, DataChannelSend := 6, PaperInject := 7, PaperInjectRetry := 8, DoNotReleaseItems := 9, DoublePaperWarning := 10, MAX_E_ALM_PBC);
END_TYPE

TYPE E_STOPREASON : (None, StopByCommand, StopBySaber, StopByManual, MAX_STOPREASON);
END_TYPE

TYPE T_Ctrl_SIf_PBC : STRUCT
  Cfg : T_Ctrl_SIf_PBC_Cfg;  (* configuration *)
  Par : T_Ctrl_SIf_PBC_Par;  (* parameter *)
  Cur : T_Ctrl_SIf_PBC_Cur;  (* current values *)
  In : T_Ctrl_SIf_PBC_In;  (* io input *)
  Out : T_Ctrl_SIf_PBC_Out;  (* io output *)
  Alm : ARRAY[1..E_ALM_PBC.MAX_E_ALM_PBC] OF T_Ctrl_Alm;  (* alarm number used in this controller *)
  Ilk : T_Ctrl_SIf_PBC_Ilk;  (* interlock of output/movements *)
END_STRUCT;
END_TYPE

TYPE T_Ctrl_SIf_PBC_Cfg : STRUCT
  bolUseTurnTableSensorForEject : BOOL;  (* True : Use the turn table sensor to detect ejects. *)
  bolEnableDataChannel : BOOL;  (* Enable the Data Channel to Saber to send the read barcodes to Saber *)
  bolGranulatAirPressureUnitAvailable : BOOL;  (* Airpressure unit for the granulate available *)
  bolEnableSaberStopDeStack : BOOL;  (* Enable or Disable the Saber Stop DeStack to do manual operation *)
END_STRUCT;
END_TYPE

TYPE T_Ctrl_SIf_PBC_Cur : STRUCT
  intPaperInBufferCount : INT;  (* How many papers are in the buffer. -1 = Paper count unknown *)
  uinPaperToEjectParameter : UINT;  (* Last Paper to eject count parameter *)
  uinPaperToEjectCount : UINT;  (* Actual count of the paper ejected *)
  uinSheetToSheetTime : UINT;  (* [ms] Time from sheet to sheet ejection in multi eject mode. *)
  bolPaperBeforeEjectAvailable : BOOL;  (* Was paper before Eject available *)
  uinPaperToPaperTime_ms : UINT;  (* Paper to paper Timeout *)
  udiLastBarcode : UDINT;  (* Last Read Barcode *)
  udiBarcodeChanged : UDINT;  (* Total Paper Counter / Also used to signal a new Barcode read. *)
END_STRUCT;
END_TYPE

TYPE T_Ctrl_SIf_PBC_Ilk : STRUCT

END_STRUCT;
END_TYPE

TYPE T_Ctrl_SIf_PBC_In : STRUCT
  bolPaperAvailableExit : BASE_PLC.T_Ctrl_IoBool;  (* This sensor shows if the buffer reaches his capacity limits *)
  bolPaperAvailableEntry : BASE_PLC.T_Ctrl_IoBool;  (* Shows if there is paper available in the buffer *)
  bolCapacityReached : BASE_PLC.T_Ctrl_IoBool;  (* Shows if there is a paper on the output of the buffer *)
  bolDoublePaperDetection : BASE_PLC.T_Ctrl_IoBool;  (* Double paper detection *)
  bolTurnTableMiddleSensor : BASE_PLC.T_Ctrl_IoBool;  (* Turn Table Mid Sensor *)
  bolAirPressorOk : BASE_PLC.T_Ctrl_IoBool;  (* Airpressure Ok *)
END_STRUCT;
END_TYPE

TYPE T_Ctrl_SIf_PBC_Out : STRUCT
  bolAirOn : BASE_PLC.T_Ctrl_IoBool;  (* Air on the Airpressure supply unit on: *)
END_STRUCT;
END_TYPE

TYPE T_Ctrl_SIf_PBC_Par : STRUCT
  udiPaperTransportTime : UDINT;  (* [ms] Paper transport timeout - Time that paper is allowed to have for the transport to the front. *)
  udiSheetToEject : UDINT;  (* Sheet to output with one run command. 0 = endless until stop *)
  udiSheetToSheetTime : UDINT;  (* [ms] Time from sheet to sheet ejection in multi eject mode in Auto Mode. *)
  udiManualSheetToSheetTime_ms : UDINT;  (* [ms] Time from sheet to sheet ejection in multi eject mode in Manual Mode. *)
  udiSimPaperTransportTime : UDINT;  (* [ms] Paper transport time simulation *)
  udiSimPaperToPaperTransportTime : UDINT;  (* [ms] Paper to paper transport time simulation *)
  udiPaperInjectRetries : UDINT;  (* # of retries for paper transport. *)
  bolEnableDoublePaperDetection : BOOL;  (* Enable Double Paper detection *)
  udiDoublePaperDebounceTime_ms : UDINT;  (* [ms] Double Paper detection sensor debounce time *)
  udiPaperInjectRetryPauseTime_ms : UDINT;  (* [ms] Retry Pause Time *)
  bolAutomaticMode : BOOL;  (* Automatic or Manual DeStacking Mode *)
  bolStopReleaseItems : BOOL;  (* Indicates that the controller must not release any item but can still collect new items (RUN state). This flag is normally set by LineControl. *)
END_STRUCT;
END_TYPE

TYPE E_ALM_PCE : (PaperSensorError := 1, MAX_E_ALM_PCE);
END_TYPE

TYPE T_Ctrl_SIf_PCE : STRUCT
  Cfg : T_Ctrl_SIf_PCE_Cfg;  (* configuration *)
  Par : T_Ctrl_SIf_PCE_Par;  (* parameter *)
  Cur : T_Ctrl_SIf_PCE_Cur;  (* current values *)
  In : T_Ctrl_SIf_PCE_In;  (* io input *)
  Out : T_Ctrl_SIf_PCE_Out;  (* io output *)
  Alm : ARRAY[1..MAX_E_ALM_PCE] OF T_Ctrl_Alm;  (* alarm number used in this controller *)
  Ilk : T_Ctrl_SIf_PCE_Ilk;  (* interlock of output/movements *)
END_STRUCT;
END_TYPE

TYPE T_Ctrl_SIf_PCE_Cfg : STRUCT

END_STRUCT;
END_TYPE

TYPE T_Ctrl_SIf_PCE_Cur : STRUCT
  uinBeltSpeed : UINT;  (* [mm/s] Belt speed *)
END_STRUCT;
END_TYPE

TYPE T_Ctrl_SIf_PCE_Ilk : STRUCT

END_STRUCT;
END_TYPE

TYPE T_Ctrl_SIf_PCE_In : STRUCT
  bolPaperAvailable : BASE_PLC.T_Ctrl_IoBool;  (* 0 = Paper not here; 1 = Paper detected *)
END_STRUCT;
END_TYPE

TYPE T_Ctrl_SIf_PCE_Out : STRUCT
  bolVacuumValveIn : BASE_PLC.T_Ctrl_IoBool;  (* Paper Incoming Belt - 0 = Vacuum Valve Closed; 1 = Vacuum valve open *)
  bolVacuumValveOut : BASE_PLC.T_Ctrl_IoBool;  (* Paper Outgoing Belt - 0 = Vacuum Valve Closed; 1 = Vacuum valve open *)
END_STRUCT;
END_TYPE

TYPE T_Ctrl_SIf_PCE_Par : STRUCT
  uinPaperEntryDelayTime_ms : UDINT;  (* [ms] Paper entry delay time. Time delay between detection and switching the vacuum *)
  uinPaperExitTime_ms : UDINT;  (* [ms] Paper exit time *)
  uinSimPaperExitTime_ms : UDINT;  (* [ms] Simulation Paper exit time *)
END_STRUCT;
END_TYPE

TYPE E_ALM_PST : (StackIncomplete := 1, NeedsEjectCommand := 2, StackOkButLastCodeNotRight := 3, StackNotOkButLastCodeRight := 4, ReadingBarcodeFailedAfterXRetries := 5, NewPaperDetectedDuringEjecting := 6, NewPaperDetectedWhileBarcodeReading := 7, MAX_E_ALM_PST) UDINT;
END_TYPE

TYPE T_Ctrl_SIf_PST : STRUCT
  Cfg : T_Ctrl_SIf_PST_Cfg;  (* configuration *)
  Par : T_Ctrl_SIf_PST_Par;  (* parameter *)
  Cur : T_Ctrl_SIf_PST_Cur;  (* current values *)
  In : T_Ctrl_SIf_PST_In;  (* io input *)
  Alm : ARRAY[1..E_ALM_PST.MAX_E_ALM_PST] OF T_Ctrl_Alm;  (* alarm number used in this controller *)
END_STRUCT;
END_TYPE

TYPE T_Ctrl_SIf_PST_Cfg : STRUCT
  bolEnableDataChannel : BOOL;  (* Enable data channel to saber *)
  uinNumOfRetryRead : UINT;  (* Number of retry barcode read command if failed *)
  usiEjectingDirection : INT;  (* Rotation direction for ejecting LEFT = 1 RIGHT = 2 *)
  usiReverseDirection : INT;  (* Rotation direction for reverse LEFT = 1 RIGHT = 2 *)
  bolEnablePstEjectControl : BOOL;  (* Enable PST controlled Eject *)
END_STRUCT;
END_TYPE

TYPE T_Ctrl_SIf_PST_Cur : STRUCT
  uinStackHight : UINT;  (* # of papers in the stack *)
  udiNumOfStacksEjectedTotal : UDINT;  (* Total number of stacks ejected *)
  bolStackIncomplete : BOOL;  (* Indicates that the last stacking job was incomplete. Run command not possible. Needs eject command from saber. *)
END_STRUCT;
END_TYPE

TYPE T_Ctrl_SIf_PST_In : STRUCT
  bolSensorPaperAtOperatorPos : BASE_PLC.T_Ctrl_IoBoolDebounced;  (* Sensor detects if a paper is at the operator position *)
  bolSensorStopperPosition : BASE_PLC.T_Ctrl_IoBoolDebounced;  (* Sensor detects the stopper position (TRUE = stopper position down , FALSE = stopper position up) *)
  bolSensorOutfeed : BASE_PLC.T_Ctrl_IoBoolDebounced;  (* Sensor detects paper on outfeed position *)
  bolSensorInfeed : BASE_PLC.T_Ctrl_IoBool;  (* Sensor detects paper on infeed position *)
END_STRUCT;
END_TYPE

TYPE T_Ctrl_SIf_PST_Par : STRUCT
  uinStackHight : UINT;  (* Stack hight in # of paper to eject. Sent by saber. *)
  uliLastBarCodeInStack : ULINT;  (* Last barcode in stack. Sent by saber. If stack hight is reached and last barcode in stack detected, stacker automatically eject the whole stack. *)
  uinBeltReverseSpeed_mmsec : UINT;  (* [mm/s] Belt reverse speed to bring stopper back to up position *)
  uinBeltEjectSpeed_mmsec : UINT;  (* [mm/s] Belt speed for ejecting the whole stack *)
  udiPaperAtOpPosDebounceTime_ms : UDINT;  (* [ms] Paper is at operator position delay time *)
  udiStopperPosDebounceTime_ms : UDINT;  (* [ms] Stopper position delay time *)
  udiSensorOutfeedDebounceTime_ms : UDINT;  (* [ms] Outfeed sensor delay time *)
  udiStackEjectDelayTime_ms : UDINT;  (* [ms] Stack eject delay time - Delay before belt starts to eject the stack if hight is reached. *)
  udiStackEjectingTime_ms : UDINT;  (* [ms] Stack ejecting time - Time for how long the belt should move in eject direction *)
  udiBeltReverseDelayTime_ms : UDINT;  (* [ms] Belt reverse delay time - Delay before belt starts moving backward after ejecting stack. *)
  udiBarcodeReaderTriggerDelayTime_ms : UDINT;  (* [ms] Barcode reader trigger delay time - Delay time, until a read command will be executed, after a new paper was detected at infeed sensor. *)
  udiSimTimePaperInfeedStroke_ms : UDINT;  (* [ms] Simulation time paper infeed stroke *)
END_STRUCT;
END_TYPE

{attribute 'enable_dynamic_creation'}
TYPE T_ItemPaperInfo : STRUCT
  uinPosInStack : UINT;  (* Position in the stack *)
  uliBarCode : ULINT;  (* Barcode of the paper *)
END_STRUCT;
END_TYPE

TYPE E_ALM_PTS : (PaperTransport := 1, ModeParameter := 2, TurnTableConfigMissmatch := 3, MAX_E_ALM_PTS);
END_TYPE

TYPE E_PTS_MODE : (Automatic := -2, Distribute := -1, FixA := 0, FixB := 1, FixC := 2, MAX_E_PTS_MODE);
END_TYPE

TYPE T_Ctrl_SIf_PTS : STRUCT
  Cfg : T_Ctrl_SIf_PTS_Cfg;  (* configuration *)
  Par : T_Ctrl_SIf_PTS_Par;  (* parameter *)
  Cur : T_Ctrl_SIf_PTS_Cur;  (* current values *)
  In : T_Ctrl_SIf_PTS_In;  (* io input *)
  Out : T_Ctrl_SIf_PTS_Out;  (* io output *)
  Alm : ARRAY[1..MAX_E_ALM_PTS] OF T_Ctrl_Alm;  (* alarm number used in this controller *)
  Ilk : T_Ctrl_SIf_PTS_Ilk;  (* interlock of output/movements *)
END_STRUCT;
END_TYPE

TYPE T_Ctrl_SIf_PTS_Cfg : STRUCT
  bolBarcodeReaderAvailable : BOOL;  (* Turns the barcode reader intelligence on. This makes the PTS nearly self sustained. *)
  bolEntrySensorAvailable : BOOL;  (* If there is no barcode but a sensor at the end of the entry belt *)
  aFixPosDef : ARRAY[0..(E_PTS_MODE.MAX_E_PTS_MODE - 1)] OF T_PTS_InOutPositions;  (* Paper Input and Ouput Positions for the fixed modes *)
  aAutoPosDef : ARRAY[0..(cPTS_MAX_AUTOPOS - 1)] OF T_PTS_InOutPositions;  (* Automatic Mode Input and Output Positions *)
  aDefaultAutoPos : UINT;  (* Automatic Mode Default Input Positions *)
  aDistributionPositionDefinition : ARRAY[0..(PTS_CmdState.cPTS_MAX_DISTRIBUTION - 1)] OF E_PTS_MODE;  (* Paper Input and Ouput Positions for the fixed modes *)
  bolPositionMalteserEnable : BOOL;  (* Start positioning the malteser wheel before turning *)
  bolRaxEnable : BOOL;  (* Use Servo Axis instead of Malteser for turning *)
END_STRUCT;
END_TYPE

TYPE T_Ctrl_SIf_PTS_Cur : STRUCT
  rInOutPosition : T_PTS_InOutPositions;  (* Actual Sheet In- Out- Positions *)
  iActualDistributionIndex : INT;  (* Saves the last executed distribution index *)
  udiPaperInTurnDelayTime : UDINT;  (* [ms] Time to wait after paper was detected before to turn. *)
  udiPaperOutTurnDelayTime : UDINT;  (* [ms] Time to wait after paper is not detected anymore before to turn back. *)
  udiPTS_Counter : UDINT;  (* Count of turn movements in long term test *)
END_STRUCT;
END_TYPE

TYPE T_Ctrl_SIf_PTS_Ilk : STRUCT

END_STRUCT;
END_TYPE

TYPE T_Ctrl_SIf_PTS_In : STRUCT
  bolPaperAvailable : BASE_PLC.T_Ctrl_IoBool;  (* This sensor shows if the paper is at the middle table possition *)
  bolPaperAtBeltExit : BASE_PLC.T_Ctrl_IoBool;  (* This sensor shows if the paper is available at the exit of the input belt *)
END_STRUCT;
END_TYPE

TYPE T_Ctrl_SIf_PTS_Out : STRUCT

END_STRUCT;
END_TYPE

TYPE T_Ctrl_SIf_PTS_Par : STRUCT
  udiPaperInTurnDelayTime : UDINT;  (* [ms] Time to wait after paper was detected before to turn. *)
  udiPaperOutTurnDelayTime : UDINT;  (* [ms] Time to wait after paper is not detected anymore before to turn back. *)
  udiPaperBarcodeToInputSensorTime : UDINT;  (* [ms] Timeout for the time the Paper can have between Barcode reader and Paper on table sensor. *)
  eMode : E_PTS_MODE;  (* Mode for turning *)
  udiSimPaperBarcodeToInputSensorTime : UDINT;  (* [ms] Simulation Timeout for the time the Paper can have between Barcode reader and Paper on table sensor. *)
  bolLongTimeTestEnable : BOOL;  (* Activate long time test *)
END_STRUCT;
END_TYPE

TYPE T_PTS_InOutPositions : STRUCT
  uinInput : UINT;
  uinOutput : UINT;
  eDirection : E_TURN_DIRECTION;
END_STRUCT;
END_TYPE

TYPE T_GRR : STRUCT
  io : T_GRR_IO;
  ctrl : T_GRR_CTRL;
  id : T_GRR_ID;
END_STRUCT;
END_TYPE

TYPE T_GRR_CTRL : STRUCT
  fbGrr : FB_GRR;
END_STRUCT;
END_TYPE

TYPE T_GRR_ID : STRUCT
  Grr : INT;
END_STRUCT;
END_TYPE

TYPE T_GRR_IO : STRUCT
  Out_intCommand : REFERENCE TO REFERENCE TO INT;
  Out_intConveyorBelt : REFERENCE TO REFERENCE TO INT;
  Out_intPowderVibrator : REFERENCE TO REFERENCE TO INT;
  Out_intConveyorVibrator : REFERENCE TO REFERENCE TO INT;
  Out_intAnalogValue : REFERENCE TO REFERENCE TO INT;
  Out_uinFilterClearingCycleTime_min : REFERENCE TO REFERENCE TO UINT;
  Out_bolToggleBitGrr : REFERENCE TO REFERENCE TO BOOL;
  In_bolSystemOk : REFERENCE TO REFERENCE TO BOOL;
  In_bolMainPressureError : REFERENCE TO REFERENCE TO BOOL;
  In_bolEoffOrFuseOk : REFERENCE TO REFERENCE TO BOOL;
  In_bolPowderLowWarning : REFERENCE TO REFERENCE TO BOOL;
  In_bolAutoMode : REFERENCE TO REFERENCE TO BOOL;
  In_intState : REFERENCE TO REFERENCE TO INT;
  In_bolToggleBitGrn : REFERENCE TO REFERENCE TO BOOL;
  In_intMainPressure : REFERENCE TO REFERENCE TO INT;
END_STRUCT;
END_TYPE

TYPE T_JCL : STRUCT
  io : T_JCL_IO;
  ctrl : T_JCL_CTRL;
  id : T_JCL_ID;
END_STRUCT;
END_TYPE

TYPE T_JCL_CTRL : STRUCT
  fbJcl : FB_JCL;
  fbJcl_Tcp : FB_TCP;
END_STRUCT;
END_TYPE

TYPE T_JCL_ID : STRUCT
  Jcl : INT;
  Jcl_Tcp : INT;
END_STRUCT;
END_TYPE

TYPE T_JCL_IO : STRUCT

END_STRUCT;
END_TYPE

TYPE T_BCH : STRUCT
  io : T_BCH_IO;
  ctrl : T_BCH_CTRL;
  id : T_BCH_ID;
  datachn : T_BCH_DATACHN;
END_STRUCT;
END_TYPE

TYPE T_BCH_CTRL : STRUCT
  fbBch : FB_BCH;
  fbBch_Bcc : FB_BCC;
  fbBch_Bcc_Bcd : FB_BCD;
END_STRUCT;
END_TYPE

TYPE T_BCH_DATACHN : STRUCT
  rSendData : T_IdBaseSendData;
END_STRUCT;
END_TYPE

TYPE T_BCH_ID : STRUCT
  Bch : INT;
  Bch_Bcc : INT;
  Bch_Bcc_Bcd : INT;
END_STRUCT;
END_TYPE

TYPE T_BCH_IO : STRUCT
  In_bolSensorTrigScan : REFERENCE TO REFERENCE TO BOOL;
END_STRUCT;
END_TYPE

TYPE T_OVN : STRUCT
  io : T_OVN_IO;
  ctrl : T_OVN_CTRL;
  id : T_OVN_ID;
  datachn : T_OVN_DATACHN;
END_STRUCT;
END_TYPE

TYPE T_OVN_CTRL : STRUCT
  fbOvn : FB_OVN;
  fbOvn_Ibh : FB_IBH;
END_STRUCT;
END_TYPE

TYPE T_OVN_DATACHN : STRUCT
  rSendData : T_OvenSendData;
END_STRUCT;
END_TYPE

TYPE T_OVN_ID : STRUCT
  Ovn : INT;
  Ovn_Ibh : INT;
END_STRUCT;
END_TYPE

TYPE T_OVN_IO : STRUCT
  Out_uinBcrOvenAEvent : REFERENCE TO REFERENCE TO UINT;
  Out_udiBcrOvenACode : REFERENCE TO REFERENCE TO ULINT;
  Out_uinBcrOvenBEvent : REFERENCE TO REFERENCE TO UINT;
  Out_udiBcrOvenBCode : REFERENCE TO REFERENCE TO ULINT;
  In_bolBcrDistributionTrigger : REFERENCE TO REFERENCE TO BOOL;
  In_udiBarcode_new_1 : REFERENCE TO REFERENCE TO ULINT;
  In_udiBarcode_new_2 : REFERENCE TO REFERENCE TO ULINT;
  In_uinNew_element_1 : REFERENCE TO REFERENCE TO UINT;
  In_uinNew_element_2 : REFERENCE TO REFERENCE TO UINT;
  In_udiBarcode_delete_1 : REFERENCE TO REFERENCE TO ULINT;
  In_udiBarcode_delete_2 : REFERENCE TO REFERENCE TO ULINT;
  In_uinDelete_element_1 : REFERENCE TO REFERENCE TO UINT;
  In_uinDelete_element_2 : REFERENCE TO REFERENCE TO UINT;
END_STRUCT;
END_TYPE

TYPE T_PTA : STRUCT
  io : T_PTA_IO;
  ctrl : T_PTA_CTRL;
  id : T_PTA_ID;
END_STRUCT;
END_TYPE

TYPE T_PTA_CTRL : STRUCT
  fbPta : FB_PTB;  (* PTA is a special type of PTB *)
  fbPta_Umc : FB_UMC;
END_STRUCT;
END_TYPE

TYPE T_PTA_ID : STRUCT
  Pta : INT;
  Pta_Umc : INT;
END_STRUCT;
END_TYPE

TYPE T_PTA_IO : STRUCT
  In_bolInputSensor : REFERENCE TO REFERENCE TO BOOL;
  In_bolOutputSensor : REFERENCE TO REFERENCE TO BOOL;
  In_uinUmc_Status : REFERENCE TO REFERENCE TO UINT;
  In_uinUmc_ActualSpeed : REFERENCE TO REFERENCE TO UINT;
  In_uinUmc_SetSpeed : REFERENCE TO REFERENCE TO UINT;
  In_uinUmc_IOData1 : REFERENCE TO REFERENCE TO WORD;
  In_uinUmc_ECatState : REFERENCE TO REFERENCE TO UINT;
  In_strUmc_ECatNetId : REFERENCE TO REFERENCE TO AMSNETID;
  In_uinUmc_ECatPort : REFERENCE TO REFERENCE TO WORD;
  Out_uinUmc_Control : REFERENCE TO REFERENCE TO UINT;
  Out_uinUmc_SetSpeed : REFERENCE TO REFERENCE TO UINT;
END_STRUCT;
END_TYPE

TYPE T_Belt_Cfg_Base : STRUCT
  intForwardDirection : INT;  (* Assign the motor rotation to a belt direction. *)
  intBackwardDirection : INT;  (* Assign the motor rotation to a belt direction. *)
  reaRpmDistance_mm : REAL;  (* [mm] the belt travels per motor rotation *)
END_STRUCT;
END_TYPE

TYPE T_Belt_Cur_Base : STRUCT
  uinBeltSpeed_mms : UINT;  (* [mm/s] Belt speed *)
  uinBeltSpeed_rpm : UINT;  (* [rpm] Belt speed *)
END_STRUCT;
END_TYPE

TYPE T_Belt_Par_Base : STRUCT
  uinBeltSpeed : UINT;  (* eSpeedControlSelection.EFFECTIVE_SPEED : [mm/sec] Target speed. Uses reaRpmDistance_mm and uinLC11 to calculate the rpm *)
  uinStackSpeed : UINT;  (* eSpeedControlSelection.EFFECTIVE_SPEED : [mm/sec] Target speed. Uses reaRpmDistance_mm and uinLC11 to calculate the rpm *)
END_STRUCT;
END_TYPE

TYPE T_PTB : STRUCT
  io : T_PTB_IO;
  ctrl : T_PTB_CTRL;
  id : T_PTB_ID;
END_STRUCT;
END_TYPE

TYPE T_PTB_CTRL : STRUCT
  fbPtb : FB_PTB;
  fbPtb_Umc : FB_UMC;
  fbPtb_Vpc : FB_VPC;
END_STRUCT;
END_TYPE

TYPE T_PTB_ID : STRUCT
  Ptb : INT;
  Ptb_Umc : INT;
  Ptb_Vpc : INT;
END_STRUCT;
END_TYPE

TYPE T_PTB_IO : STRUCT
  In_bolInputSensor : REFERENCE TO REFERENCE TO BOOL;
  In_bolOutputSensor : REFERENCE TO REFERENCE TO BOOL;
  In_bolVpc_VacuumSensor : REFERENCE TO REFERENCE TO BOOL;
  In_bolVpc_PumpOk : REFERENCE TO REFERENCE TO BOOL;
  Out_bolVpc_PumpOn : REFERENCE TO REFERENCE TO BOOL;
  In_bolUmc_EmoOk : REFERENCE TO REFERENCE TO BOOL;
  In_uinUmc_Status : REFERENCE TO REFERENCE TO UINT;
  In_uinUmc_ActualSpeed : REFERENCE TO REFERENCE TO UINT;
  In_uinUmc_SetSpeed : REFERENCE TO REFERENCE TO UINT;
  In_uinUmc_IOData1 : REFERENCE TO REFERENCE TO WORD;
  In_uinUmc_ECatState : REFERENCE TO REFERENCE TO UINT;
  In_strUmc_ECatNetId : REFERENCE TO REFERENCE TO AMSNETID;
  In_uinUmc_ECatPort : REFERENCE TO REFERENCE TO WORD;
  Out_uinUmc_Control : REFERENCE TO REFERENCE TO UINT;
  Out_uinUmc_SetSpeed : REFERENCE TO REFERENCE TO UINT;
END_STRUCT;
END_TYPE

TYPE T_PBC : STRUCT
  io : T_PBC_IO;
  ctrl : T_PBC_CTRL;
  id : T_PBC_ID;
END_STRUCT;
END_TYPE

TYPE T_PBC_CTRL : STRUCT
  fbPbc_PtbDeStacker : FB_PTB;
  fbPbc_PtbDeStacker_Umc : FB_UMC;
  fbPbc_PtbBelt : FB_PTB;
  fbPbc_PtbBelt_Umc : FB_UMC;
  fbPbc_PtbBelt_Vpc : FB_VPC;
  fbPbc : FB_PBC;
END_STRUCT;
END_TYPE

TYPE T_PBC_ID : STRUCT
  Pbc : INT;
  Pbc_PtbDeStacker : INT;
  Pbc_PtbDeStacker_Umc : INT;
  Pbc_PtbBelt : INT;
  Pbc_PtbBelt_Umc : INT;
  Pbc_PtbBelt_Vpc : INT;
END_STRUCT;
END_TYPE

TYPE T_PBC_IO : STRUCT
  In_bolPts_PaperSensor : REFERENCE TO REFERENCE TO BOOL;  (* TODO: describe why this is here *)
  In_bolInputSensor : REFERENCE TO REFERENCE TO BOOL;
  In_bolOutputSensor : REFERENCE TO REFERENCE TO BOOL;
  In_bolCapacitySensor : REFERENCE TO REFERENCE TO BOOL;
  In_bolDoublePaperSensor : REFERENCE TO REFERENCE TO BOOL;
  In_bolAirPressureOk : REFERENCE TO REFERENCE TO BOOL;
  Out_bolAirPressureOn : REFERENCE TO REFERENCE TO BOOL;
  In_bolPtbBelt_Vpc_VacuumSensor : REFERENCE TO REFERENCE TO BOOL;
  In_bolPtbBelt_Vpc_PumpOk : REFERENCE TO REFERENCE TO BOOL;
  Out_bolPtbBelt_Vpc_PumpOn : REFERENCE TO REFERENCE TO BOOL;
  In_uinPtbBelt_Umc_Status : REFERENCE TO REFERENCE TO UINT;
  In_uinPtbBelt_Umc_ActualSpeed : REFERENCE TO REFERENCE TO UINT;
  In_uinPtbBelt_Umc_SetSpeed : REFERENCE TO REFERENCE TO UINT;
  In_uinPtbBelt_Umc_IOData1 : REFERENCE TO REFERENCE TO WORD;
  In_uinPtbBelt_Umc_ECatState : REFERENCE TO REFERENCE TO UINT;
  In_strPtbBelt_Umc_ECatNetId : REFERENCE TO REFERENCE TO AMSNETID;
  In_uinPtbBelt_Umc_ECatPort : REFERENCE TO REFERENCE TO WORD;
  Out_uinPtbBelt_Umc_Control : REFERENCE TO REFERENCE TO UINT;
  Out_uinPtbBelt_Umc_SetSpeed : REFERENCE TO REFERENCE TO UINT;
  In_uinPtbDeStacker_Umc_Status : REFERENCE TO REFERENCE TO UINT;
  In_uinPtbDeStacker_Umc_ActualSpeed : REFERENCE TO REFERENCE TO UINT;
  In_uinPtbDeStacker_Umc_SetSpeed : REFERENCE TO REFERENCE TO UINT;
  In_uinPtbDeStacker_Umc_IOData1 : REFERENCE TO REFERENCE TO WORD;
  In_uinPtbDeStacker_Umc_ECatState : REFERENCE TO REFERENCE TO UINT;
  In_strPtbDeStacker_Umc_ECatNetId : REFERENCE TO REFERENCE TO AMSNETID;
  In_uinPtbDeStacker_Umc_ECatPort : REFERENCE TO REFERENCE TO WORD;
  Out_uinPtbDeStacker_Umc_Control : REFERENCE TO REFERENCE TO UINT;
  Out_uinPtbDeStacker_Umc_SetSpeed : REFERENCE TO REFERENCE TO UINT;
END_STRUCT;
END_TYPE

TYPE T_PCE : STRUCT
  io : T_PCE_IO;
  ctrl : T_PCE_CTRL;
  id : T_PCE_ID;
END_STRUCT;
END_TYPE

TYPE T_PCE_CTRL : STRUCT
  fbPce : FB_PCE;
  fbPce_PtbIn : FB_PTB;
  fbPce_PtbIn_Umc : FB_UMC;
  fbPce_PtbIn_Vpc : FB_VPC;
  fbPce_PtbOut : FB_PTB;
  fbPce_PtbOut_Umc : FB_UMC;
END_STRUCT;
END_TYPE

TYPE T_PCE_ID : STRUCT
  Pce : INT;
  Pce_PtbIn : INT;
  Pce_PtbIn_Umc : INT;
  Pce_PtbIn_Vpc : INT;
  Pce_PtbOut : INT;
  Pce_PtbOut_Umc : INT;
END_STRUCT;
END_TYPE

TYPE T_PCE_IO : STRUCT
  In_bolInputSensor : REFERENCE TO REFERENCE TO BOOL;
  In_bolOutputSensor : REFERENCE TO REFERENCE TO BOOL;
  In_bolCornerSensor : REFERENCE TO REFERENCE TO BOOL;
  Out_bolVacuumValveIn : REFERENCE TO REFERENCE TO BOOL;
  Out_bolVacuumValveOut : REFERENCE TO REFERENCE TO BOOL;
  In_uinUmcIn_Status : REFERENCE TO REFERENCE TO UINT;
  In_uinUmcIn_ActualSpeed : REFERENCE TO REFERENCE TO UINT;
  In_uinUmcIn_SetSpeed : REFERENCE TO REFERENCE TO UINT;
  In_uinUmcIn_IOData1 : REFERENCE TO REFERENCE TO WORD;
  In_uinUmcIn_ECatState : REFERENCE TO REFERENCE TO UINT;
  In_strUmcIn_ECatNetId : REFERENCE TO REFERENCE TO AMSNETID;
  In_uinUmcIn_ECatPort : REFERENCE TO REFERENCE TO WORD;
  Out_uinUmcIn_Control : REFERENCE TO REFERENCE TO UINT;
  Out_uinUmcIn_SetSpeed : REFERENCE TO REFERENCE TO UINT;
  In_uinUmcOut_Status : REFERENCE TO REFERENCE TO UINT;
  In_uinUmcOut_ActualSpeed : REFERENCE TO REFERENCE TO UINT;
  In_uinUmcOut_SetSpeed : REFERENCE TO REFERENCE TO UINT;
  In_uinUmcOut_IOData1 : REFERENCE TO REFERENCE TO WORD;
  In_uinUmcOut_ECatState : REFERENCE TO REFERENCE TO UINT;
  In_strUmcOut_ECatNetId : REFERENCE TO REFERENCE TO AMSNETID;
  In_uinUmcOut_ECatPort : REFERENCE TO REFERENCE TO WORD;
  Out_uinUmcOut_Control : REFERENCE TO REFERENCE TO UINT;
  Out_uinUmcOut_SetSpeed : REFERENCE TO REFERENCE TO UINT;
  In_bolVpc_VacuumSensor : REFERENCE TO REFERENCE TO BOOL;
  In_bolVpc_PumpOk : REFERENCE TO REFERENCE TO BOOL;
  Out_bolVpc_PumpOn : REFERENCE TO REFERENCE TO BOOL;
END_STRUCT;
END_TYPE

TYPE T_PST : STRUCT
  io : T_PST_IO;
  ctrl : T_PST_CTRL;
  id : T_PST_ID;
END_STRUCT;
END_TYPE

TYPE T_PST_CTRL : STRUCT
  fbPst : FB_PST;
  fbPst_Ptb : FB_PTB;
  fbPst_Ptb_Umc : FB_UMC;
  fbPst_Ptb_Vpc : FB_VPC;
END_STRUCT;
END_TYPE

TYPE T_PST_ID : STRUCT
  Pst : INT;
  Pst_Ptb : INT;
  Pst_Ptb_Umc : INT;
  Pst_Ptb_Vpc : INT;
END_STRUCT;
END_TYPE

TYPE T_PST_IO : STRUCT
  In_bolSensorPaperAtOperatorPos : REFERENCE TO REFERENCE TO BOOL;
  In_bolSensorStopperPosition : REFERENCE TO REFERENCE TO BOOL;
  In_bolSensorInfeed : REFERENCE TO REFERENCE TO BOOL;
  In_bolSensorOutfeed : REFERENCE TO REFERENCE TO BOOL;
  In_bolPtb_InputSensor : REFERENCE TO REFERENCE TO BOOL;
  In_bolPtb_OutputSensor : REFERENCE TO REFERENCE TO BOOL;
  In_bolPtb_Vpc_VacuumSensor : REFERENCE TO REFERENCE TO BOOL;
  In_bolPtb_Vpc_PumpOk : REFERENCE TO REFERENCE TO BOOL;
  Out_bolPtb_Vpc_PumpOn : REFERENCE TO REFERENCE TO BOOL;
  In_uinPtb_Umc_Status : REFERENCE TO REFERENCE TO UINT;
  In_uinPtb_Umc_ActualSpeed : REFERENCE TO REFERENCE TO UINT;
  In_uinPtb_Umc_SetSpeed : REFERENCE TO REFERENCE TO UINT;
  In_uinPtb_Umc_IOData1 : REFERENCE TO REFERENCE TO WORD;
  In_uinPtb_Umc_ECatState : REFERENCE TO REFERENCE TO UINT;
  In_strPtb_Umc_ECatNetId : REFERENCE TO REFERENCE TO AMSNETID;
  In_uinPtb_Umc_ECatPort : REFERENCE TO REFERENCE TO WORD;
  Out_uinPtb_Umc_Control : REFERENCE TO REFERENCE TO UINT;
  Out_uinPtb_Umc_SetSpeed : REFERENCE TO REFERENCE TO UINT;
END_STRUCT;
END_TYPE

TYPE T_PTS : STRUCT
  io : T_PTS_IO;
  ctrl : T_PTS_CTRL;
  id : T_PTS_ID;
END_STRUCT;
END_TYPE

TYPE T_PTS_CTRL : STRUCT
  fbPts_RAX_POD : FB_POD;
  fbPts_RAX : FB_RAX;
  fbPts_Ptb : FB_PTB;
  fbPts_Ptb_Umc : FB_UMC;
  fbPts_Ptb_Vpc : FB_VPC;
  fbPts_Mdc_Umc : FB_UMC;
  fbPts_Mdc : FB_MDC;
  fbPts : FB_PTS;
END_STRUCT;
END_TYPE

TYPE T_PTS_ID : STRUCT
  Pts : INT;
  Pts_Ptb : INT;
  Pts_Ptb_Umc : INT;
  Pts_Ptb_Vpc : INT;
  Pts_Mdc : INT;
  Pts_Mdc_Umc : INT;
  Pts_RAX_POD : INT;  (* New Servo Drive PLC opend driver *)
  Pts_RAX : INT;  (* New Servo Drive *)
END_STRUCT;
END_TYPE

TYPE T_PTS_IO : STRUCT
  In_bolPaperSensor : REFERENCE TO REFERENCE TO BOOL;
  In_bolMdc_CrossPositionSensor : REFERENCE TO REFERENCE TO BOOL;
  In_bolMdc_TablePositionSensor : REFERENCE TO REFERENCE TO BOOL;
  In_uinMdc_Umc_Status : REFERENCE TO REFERENCE TO UINT;
  In_uinMdc_Umc_ActualSpeed : REFERENCE TO REFERENCE TO UINT;
  In_uinMdc_Umc_SetSpeed : REFERENCE TO REFERENCE TO UINT;
  In_uinMdc_Umc_IOData1 : REFERENCE TO REFERENCE TO WORD;
  In_uinMdc_Umc_ECatState : REFERENCE TO REFERENCE TO UINT;
  In_strMdc_Umc_ECatNetId : REFERENCE TO REFERENCE TO AMSNETID;
  In_uinMdc_Umc_ECatPort : REFERENCE TO REFERENCE TO WORD;
  Out_uinMdc_Umc_Control : REFERENCE TO REFERENCE TO UINT;
  Out_uinMdc_Umc_SetSpeed : REFERENCE TO REFERENCE TO UINT;
  In_uinPtb_Umc_Status : REFERENCE TO REFERENCE TO UINT;
  In_uinPtb_Umc_ActualSpeed : REFERENCE TO REFERENCE TO UINT;
  In_uinPtb_Umc_SetSpeed : REFERENCE TO REFERENCE TO UINT;
  In_uinPtb_Umc_IOData1 : REFERENCE TO REFERENCE TO WORD;
  In_uinPtb_Umc_ECatState : REFERENCE TO REFERENCE TO UINT;
  In_strPtb_Umc_ECatNetId : REFERENCE TO REFERENCE TO AMSNETID;
  In_uinPtb_Umc_ECatPort : REFERENCE TO REFERENCE TO WORD;
  Out_uinPtb_Umc_Control : REFERENCE TO REFERENCE TO UINT;
  Out_uinPtb_Umc_SetSpeed : REFERENCE TO REFERENCE TO UINT;
  In_bolPtb_Vpc_VacuumSensor : REFERENCE TO REFERENCE TO BOOL;
  In_bolPtb_Vpc_PumpOk : REFERENCE TO REFERENCE TO BOOL;
  Out_bolPtb_Vpc_PumpOn : REFERENCE TO REFERENCE TO BOOL;
  In_bolRax_PositionSensor : REFERENCE TO REFERENCE TO BOOL;
END_STRUCT;
END_TYPE

TYPE T_OvenSendData : STRUCT
  fbDataChannel : FB_IdBaseSendDch;
  rDataChannelItem : T_Oven_DCH;
  fbFifo : FB_DataChannelSenderFifo;
END_STRUCT;
END_TYPE

{attribute 'enable_dynamic_creation'}
TYPE T_Oven_DCH : STRUCT
  rBaseInfo : T_ItemBase;
  udiIdentification : ULINT;  (* Paper ID *)
  bTrash : BOOL;  (* Recipe process parameter -------------------------------------------------------------- Oven Data *)
  diTimeInOven_s : DINT;
  diTemperature_mc : ARRAY[0..(MAX_NUMBER_OF_OVEN_MODULES - 1)] OF DINT;
  diAirflow_prc : ARRAY[0..(MAX_NUMBER_OF_OVEN_MODULES - 1)] OF DINT;
END_STRUCT;
END_TYPE

TYPE U_JCL_Message : UNION
  Cmd : T_JCL_Command;
  State : T_JCL_State;
  PrintDone : T_JCL_PrintDone;
  ReqCleaning : T_JCL_RequestCleaning;
  AlmMsg : T_JCL_AlmMsg;
END_UNION;
END_TYPE

FUNCTION_BLOCK FB_IBH EXTENDS FB_CtrlBase
  VAR_OUTPUT
    Out_iStatus : INT;  (* Status *)
    Out_bOff : BOOL;  (* Machine off *)
    Out_bBeltOn : BOOL;  (* Band on *)
    Out_bManual : BOOL;  (* Manual Mode *)
    Out_bRun : BOOL;  (* Standart drying process *)
    Out_bSetParam : BOOL;  (* Set Parameter *)
    Out_bGetParam : BOOL;  (* Get Parameter *)
    Out_bAckError : BOOL;  (* Resetting error *)
    Out_adiTemp_dc : ARRAY[0..(MAX_NUMBER_OF_OVEN_MODULES - 1)] OF DINT;  (* Actual temperature in deci °C *)
    Out_adiAir_p : ARRAY[0..(MAX_NUMBER_OF_OVEN_MODULES - 1)] OF DINT;  (* Aactual airflow in % *)
    Out_diSpeed_mm_min : DINT;  (* Actual belt speed in mm/min *)
    Out_iErrorLevel : INT;  (* 1=Information, 2=Warning, 3=Error *)
    Out_iErrorID : INT;  (* Error ID (e.g. 100=temperature overflow) *)
    Out_bDriverConnected : BOOL;
    Out_bDriverError : BOOL;
    Out_udiDriverErrorID : UDINT;
  END_VAR
  VAR
    SIf : T_Ctrl_SIf_IBH;  (* Specific interface struct for public access *)
    iOff : INT;  (* Turns oven off *)
    iBeltOn : INT;  (* Turns belt on *)
    iManual : INT;  (* Puts oven to manual *)
    iRun : INT;  (* Standart drying process *)
    iSetParam : INT;  (* Set Parameter *)
    iGetParam : INT;  (* Get Parameter *)
    adiTemp_dc : ARRAY[0..(MAX_NUMBER_OF_OVEN_MODULES - 1)] OF DINT;  (* Temperature in deci °C *)
    adiAir_p : ARRAY[0..(MAX_NUMBER_OF_OVEN_MODULES - 1)] OF DINT;  (* Airflow in % *)
    diSpeed_mm_min : DINT;  (* Belt speed in mm/min *)
    iAckError : INT;  (* Try to reset error *)
    bIncrementSetParam : BOOL;
    bRememberIncrementSetParam : BOOL;
    fbOpen : Tc2_S5S7Com.FB_NLinkOpen;
    fbWrite : Tc2_S5S7Com.FB_NLinkWrite;
    fbFetch : Tc2_S5S7Com.FB_NLinkFetch;
    fbClose : Tc2_S5S7Com.FB_NLinkClose;
    hLink : T_HNLINK;  (* Communication link handle *)
    anReadBuffer : ARRAY[0..(READ_BUFFER_LENGTH - 1)] OF BYTE;  (* read data buffer *)
    anWriteBuffer : ARRAY[0..(WRITE_BUFFER_LENGTH - 1)] OF BYTE;  (* data to write *)
    iSimStatus : INT;  (* simulation *)
    bSimOff : BOOL;
    bSimBeltOn : BOOL;
    bSimManual : BOOL;
    bSimRun : BOOL;
  END_VAR

                  (*__________________________________________________________________________________________________
¦	
¦	Vistaprint Schweiz GmbH
¦	CH - 8401 Winterthur
¦
¦	www.vistaprint.ch - info@vistaprint.ch
¦___________________________________________________________________________________________________

Function desription:
IBH Link Connection Implementation

History:
Version		Date			Author		Comment
---------------------------------------------------------------------------------------------------
0.00.1		09.01.2014		BB			Start history
___________________________________________________________________________________________________*)

SUPER^();
                

ACTION setAckError:
                      IF (iAckError = MAX_INT OR iAckError < 0) THEN
	iAckError := 0;
END_IF

IF NOT CIf.SwCfg.bolSimulation THEN
	iAckError := iAckError + 1;
END_IF
                    
END_ACTION

ACTION setRun:
                      IF (iRun = MAX_INT OR iRun < 0) THEN
	iRun := 0;
END_IF

IF NOT CIf.SwCfg.bolSimulation THEN
	iRun := iRun + 1;
END_IF

// simulation
iSimStatus := 4;
bSimOff := FALSE;
bSimBeltOn := FALSE;
bSimManual := FALSE;
bSimRun := TRUE;
                    
END_ACTION

ACTION setOff:
                      IF (iOff = MAX_INT OR ioff < 0) THEN
	iOff := 0;
END_IF

IF NOT CIf.SwCfg.bolSimulation THEN
	iOff := iOff + 1;
END_IF

// simulation
iSimStatus := 1;
bSimOff := TRUE;
bSimBeltOn := FALSE;
bSimManual := FALSE;
bSimRun := FALSE;
                    
END_ACTION

ACTION setBeltOn:
                      IF (iBeltOn = MAX_INT OR iBeltOn < 0) THEN
	iBeltOn := 0;
END_IF

IF NOT CIf.SwCfg.bolSimulation THEN
	iBeltOn := iBeltOn + 1;
END_IF

// simulation
iSimStatus := 2;
bSimOff := FALSE;
bSimBeltOn := TRUE;
bSimManual := FALSE;
bSimRun := FALSE;
                    
END_ACTION

ACTION setStandby:
                      IF (iManual = MAX_INT OR iManual < 0) THEN
	iManual := 0;
END_IF

IF NOT CIf.SwCfg.bolSimulation THEN
	iManual := iManual + 1;
END_IF

// simulation
iSimStatus := 3;
bSimOff := FALSE;
bSimBeltOn := FALSE;
bSimManual := TRUE;
bSimRun := FALSE;
                    
END_ACTION

{attribute 'object_name' := 'sta_OFF'}
METHOD sta_OFF : BOOL
                        // state implemetation

// Entry action
//--------------------------------------------------------------------------------------
	IF (me.StateMachine.intState <> me.StateMachine.intStateLastCycle) THEN
		// state changed since last cycle
		me.StateMachine.intStateLastCycle := me.StateMachine.intState;
	END_IF

	
// Cyclic action
//--------------------------------------------------------------------------------------	
	// Simulation
	IF (CIf.SwCfg.bolSimulation) THEN
		;
	END_IF
	
	// State Change Condition
	IF CIf.SwCfg.bolEnable THEN
		CASE me.intCmd OF
			// CONNECT
			IBH_CmdState.cCMD_CONNECT, IBH_CmdState.cCMD_WRITE, IBH_CmdState.cCMD_READ:
				me.StateMachine.intStateNext := IBH_CmdState.cSTA_CONNECTBusy;
		ELSE
			// DEFAULT
			;
		END_CASE
	END_IF


// Exit action
//--------------------------------------------------------------------------------------
	IF (me.StateMachine.intState <> me.StateMachine.intStateNext) THEN
		// state is going to change
		;
	END_IF
                      
END_METHOD

{attribute 'object_name' := 'sta_PON'}
METHOD sta_PON : BOOL
                        // state implemetation

// Entry action
//--------------------------------------------------------------------------------------
	IF (me.StateMachine.intState <> me.StateMachine.intStateLastCycle) THEN
		// state changed since last cycle
		me.StateMachine.intStateLastCycle := me.StateMachine.intState;
	END_IF

	
// Cyclic action
//--------------------------------------------------------------------------------------	
	// Simulation
	IF (CIf.SwCfg.bolSimulation) THEN
		;
	END_IF
	
	// State Change Condition
	me.StateMachine.intStateNext := Base_PLC.cSTA_OFFBusy;
	

// Exit action
//--------------------------------------------------------------------------------------
	IF (me.StateMachine.intState <> me.StateMachine.intStateNext) THEN
		// state is going to change
		;
	END_IF
                      
END_METHOD

{attribute 'object_name' := 'CtrlInit'}
METHOD CtrlInit : BOOL
                        SUPER^.CtrlInit();

// add childs
// ...
                      
END_METHOD

{attribute 'object_name' := 'setTemp'}
METHOD setTemp
  VAR_INPUT
    In_adiTemp_dc : ARRAY[1..MAX_NUMBER_OF_OVEN_MODULES] OF DINT;  (* Temperature in deci °C *)
  END_VAR
                        adiTemp_dc := In_adiTemp_dc;
bIncrementSetParam := TRUE;
                      
END_METHOD

{attribute 'object_name' := 'FB_init'}
METHOD FB_init : BOOL
  VAR_INPUT
    bInitRetains : BOOL;  (* if TRUE, the retain variables are initialized (warm start / cold start) *)
    bInCopyCode : BOOL;  (* if TRUE, the instance afterwards gets moved into the copy code (online change) *)
  END_VAR
  VAR
    uiIdx : UINT;
  END_VAR
                        //------------------------------------------------------------------------------------------------------------------------
// to manually change in new FUB implementation!!!
// define valid commands for this controller
FOR uiIdx:=0 TO (SIZEOF(CIf.Job.aCmdList)/SIZEOF(CIf.Job.aCmdList[0])-1) BY 1 DO
	IF (CIf.Job.aCmdList[uiIdx].intCmd=cSTA_INITIALIZED) THEN
		// found first empty array element
		EXIT;
	END_IF
END_FOR

// Add configuration of own comands
CIf.Job.aCmdList[uiIdx].intCmd := IBH_CmdState.cCMD_CONNECT;
CIf.Job.aCmdList[uiIdx].strName := 'CONNECT';
CIf.Job.aCmdList[uiIdx].bolAvailable := TRUE;
uiIdx := uiIdx+1;
CIf.Job.aCmdList[uiIdx].intCmd := IBH_CmdState.cCMD_WRITE;
CIf.Job.aCmdList[uiIdx].strName := 'WRITE';
CIf.Job.aCmdList[uiIdx].bolAvailable := TRUE;
uiIdx := uiIdx+1;
CIf.Job.aCmdList[uiIdx].intCmd := IBH_CmdState.cCMD_READ;
CIf.Job.aCmdList[uiIdx].strName := 'READ';
CIf.Job.aCmdList[uiIdx].bolAvailable := TRUE;
uiIdx := uiIdx+1;
CIf.Job.aCmdList[uiIdx].intCmd := IBH_CmdState.cCMD_DISCONNECT;
CIf.Job.aCmdList[uiIdx].strName := 'DISCONNECT';
CIf.Job.aCmdList[uiIdx].bolAvailable := TRUE;

// set name of class/typ
CIf.Info.strType := 'FB_IBH';
CIf.Info.strFullName := 'IBH Link';

//*******************************************************************************
// initial values
//*******************************************************************************

// Software configuration
CIf.SwCfg.bolExist := TRUE;
CIf.SwCfg.bolEnable := TRUE;
CIf.SwCfg.bolSimulation := FALSE;

// Internal Variables (Input)
iOff := 0;
iBeltOn := 0;
iManual := 0;
iRun := 0;
iSetParam := 0;
iGetParam := 0;
FOR uiIdx:=0 TO MAX_NUMBER_OF_OVEN_MODULES-1 BY 1 DO
	adiTemp_dc[uiIdx] := 0;
	adiAir_p[uiIdx] := 0;
END_FOR
diSpeed_mm_min := 0;
iAckError := 0;
bIncrementSetParam := FALSE;
bRememberIncrementSetParam := FALSE;

// simulation
iSimStatus := 1;
bSimOff := TRUE;
bSimBeltOn := FALSE;
bSimManual := FALSE;
bSimRun := FALSE;

// Configuration
SIf.Cfg.tIpAddress						:= '192.168.0.50';
SIf.Cfg.udiPortAdress					:= 1099;
SIf.Cfg.nDeviceAddress					:= 2;
SIf.Cfg.nDatablockNumber				:= 22;
SIf.Cfg.tTimeout						:= T#15S;

SIf.Cfg.nWriteStartAddress				:= 0;
SIf.Cfg.nReadStartAddress				:= 110;

SIf.Cfg.uiByteOffset_rd_iStatus			:= 0;
SIf.Cfg.uiByteOffset_rd_bOff			:= 10;
SIf.Cfg.uiBitOffset_rd_bOff				:= 0;
SIf.Cfg.uiByteOffset_rd_bBeltOn			:= 10;
SIf.Cfg.uiBitOffset_rd_bBeltOn			:= 1;
SIf.Cfg.uiByteOffset_rd_bManual			:= 10;
SIf.Cfg.uiBitOffset_rd_bManual			:= 2;
SIf.Cfg.uiByteOffset_rd_bRun			:= 10;
SIf.Cfg.uiBitOffset_rd_bRun				:= 3;
SIf.Cfg.uiByteOffset_rd_bSetParam		:= 10;
SIf.Cfg.uiBitOffset_rd_bSetParam		:= 4;
SIf.Cfg.uiByteOffset_rd_bGetParam		:= 10;
SIf.Cfg.uiBitOffset_rd_bGetParam		:= 5;
SIf.Cfg.uiByteOffset_rd_bAckError		:= 10;
SIf.Cfg.uiBitOffset_rd_bAckError		:= 6;
SIf.Cfg.uiByteOffset_rd_adiTemp_mc		:= 30;
SIf.Cfg.uiByteOffset_rd_adiAir_p		:= 62;
SIf.Cfg.uiByteOffset_rd_diSpeed_mm_min	:= 94;
SIf.Cfg.uiByteOffset_rd_iErrorLevel		:= 98;
SIf.Cfg.uiByteOffset_rd_iErrorID		:= 100;
SIf.Cfg.uiByteOffset_rd_iErrorValue		:= 102;

SIf.Cfg.uiByteOffset_wr_iOff			:= 0;
SIf.Cfg.uiByteOffset_wr_iBeltOn			:= 2;
SIf.Cfg.uiByteOffset_wr_iManual			:= 4;
SIf.Cfg.uiByteOffset_wr_iRun			:= 6;
SIf.Cfg.uiByteOffset_wr_iSetParam		:= 8;
SIf.Cfg.uiByteOffset_wr_iGetParam		:= 10;
SIf.Cfg.uiByteOffset_wr_iAckError		:= 12;
SIf.Cfg.uiByteOffset_wr_adiTemp_mc		:= 30;
SIf.Cfg.uiByteOffset_wr_adiAir_p		:= 62;
SIf.Cfg.uiByteOffset_wr_diSpeed_mm_min	:= 94;
                      
END_METHOD

{attribute 'object_name' := 'sta_CONNECTBusy'}
METHOD sta_CONNECTBusy : BOOL
  VAR
    bBusy : BOOL;
    bError : BOOL;
    udiErrID : UDINT;
  END_VAR
                        // state implemetation

// Entry action
//--------------------------------------------------------------------------------------
	IF (me.StateMachine.intState <> me.StateMachine.intStateLastCycle) THEN
		// state changed since last cycle
		me.StateMachine.intStateLastCycle := me.StateMachine.intState;
		
		THIS^.fbOpen.stSettings.sHost			:= SIf.Cfg.tIpAddress; (* Remote (server) address. String containing an (Ipv4) Internet Protocol dotted address. *)
		THIS^.fbOpen.stSettings.nPort			:= SIf.Cfg.udiPortAdress; (* Remote (server) Internet Protocol (IP) port. *)
		THIS^.fbOpen.stSettings.eProtocol		:= eNLinkProtocol_MPI; (* Lan link protocol type *)
		THIS^.fbOpen.stSettings.eTransport		:= eNLinkTransport_TCPIP; (* Used transport protocol *)
		THIS^.fbOpen.tTimeout					:= SIf.Cfg.tTimeout; (* Maximum time allowed for the execution of the command *)
		
		IF NOT CIf.SwCfg.bolSimulation THEN
			// Open connection
			THIS^.fbOpen( hLink := hLink, bExecute := FALSE);
			THIS^.fbOpen( hLink := hLink, bExecute := TRUE);
		END_IF
	END_IF

	
// Cyclic action
//--------------------------------------------------------------------------------------	
	
	// check status of fbOpen
	THIS^.fbOpen( hLink := hLink, bExecute := FALSE, bBusy=>bBusy, bError=>bError, nErrID=>udiErrID);
	
	// Simulation
	IF (CIf.SwCfg.bolSimulation) THEN
		bBusy := FALSE;
		bError := FALSE;
		udiErrID := 0;
	END_IF
	
	// State Change Condition
	IF NOT bBusy THEN
		Out_udiDriverErrorID := udiErrID;
		IF bError THEN
			Out_bDriverError := TRUE;
			me.StateMachine.intStateNext := IBH_CmdState.cSTA_DISCONNECTBusy;
		ELSE
			Out_bDriverError := FALSE;
			me.StateMachine.intStateNext := IBH_CmdState.cSTA_CONNECT;
		END_IF
	END_IF


// Exit action
//--------------------------------------------------------------------------------------
	IF (me.StateMachine.intState <> me.StateMachine.intStateNext) THEN
		// state is going to change
		;
	END_IF
                      
END_METHOD

{attribute 'object_name' := 'bitAccess'}
METHOD bitAccess : BOOL
  VAR_INPUT
    in_byte : BYTE;
    in_bit : UINT;
  END_VAR
                        CASE in_bit OF
	0: bitAccess := in_byte.0;
	1: bitAccess := in_byte.1;
	2: bitAccess := in_byte.2;
	3: bitAccess := in_byte.3;
	4: bitAccess := in_byte.4;
	5: bitAccess := in_byte.5;
	6: bitAccess := in_byte.6;
	7: bitAccess := in_byte.7;
ELSE
	bitAccess := in_byte.0;
END_CASE
                      
END_METHOD

{attribute 'object_name' := 'sta_READBusy'}
METHOD sta_READBusy : BOOL
  VAR
    bBusy : BOOL;
    bError : BOOL;
    udiErrID : UDINT;
  END_VAR
                        // state implemetation

// Entry action
//--------------------------------------------------------------------------------------
	IF (me.StateMachine.intState <> me.StateMachine.intStateLastCycle) THEN
		// state changed since last cycle
		me.StateMachine.intStateLastCycle := me.StateMachine.intState;
		
		IF NOT CIf.SwCfg.bolSimulation THEN
			// Read data
			fbFetch(hLink := hLink, bExecute := FALSE );
			fbFetch(hLink := hLink, (* Communication link handle *)
					devAddr := SIf.Cfg.nDeviceAddress, (* Device address, MPI address of the remote component or its PROFIBUS address *)
					eArea:= eNLinkArea_DB, (* PLC data area *)
					nDB:= SIf.Cfg.nDatablockNumber, (* Data block number from which the data is read (DB, DX only). *)
					nOffset:= SIf.Cfg.nReadStartAddress, (* Start byte/word address from which the data are taken to *)
					cbBuffer:= SIZEOF(anReadBuffer), (* Contains the max. number of destination bytes to be received *)
					pBuffer:= ADR(anReadBuffer), (* Contains the address of the destination buffer for the received data *)
					bExecute:= TRUE); (* Rising edge at this input starts command execution *)
		END_IF
	END_IF

	
// Cyclic action
//--------------------------------------------------------------------------------------	
	
	// check status of fbFetch
	fbFetch(hLink := hLink, bExecute := FALSE, bBusy=>bBusy, bError=>bError, nErrID=>udiErrID);
	
	// Simulation
	IF (CIf.SwCfg.bolSimulation) THEN
		bBusy := FALSE;
		bError := FALSE;
		udiErrID := 0;
	END_IF
	
	// State Change Condition
	IF NOT bBusy THEN
		Out_udiDriverErrorID := udiErrID;
		IF bError THEN
			Out_bDriverError := TRUE;
			me.StateMachine.intStateNext := IBH_CmdState.cSTA_DISCONNECTBusy;
		ELSE
			Out_bDriverError := FALSE;
			me.StateMachine.intStateNext := IBH_CmdState.cSTA_READ;
		END_IF
	END_IF


// Exit action
//--------------------------------------------------------------------------------------
	IF (me.StateMachine.intState <> me.StateMachine.intStateNext) THEN
		// state is going to change
		;
	END_IF
                      
END_METHOD

{attribute 'object_name' := 'sta_WRITEBusy'}
METHOD sta_WRITEBusy : BOOL
  VAR
    uiIdx : UINT;
    bBusy : BOOL;
    bError : BOOL;
    udiErrID : UDINT;
  END_VAR
                        // state implemetation

// Entry action
//--------------------------------------------------------------------------------------
	IF (me.StateMachine.intState <> me.StateMachine.intStateLastCycle) THEN
		// state changed since last cycle
		me.StateMachine.intStateLastCycle := me.StateMachine.intState;
		
		me.SubStateMachine.intState := IBH_CmdState.cSTA_SUB_1;
		me.SubStateMachine.intStateNext := IBH_CmdState.cSTA_SUB_1;
		
		// Prepare Write Buffer
		// !!!ATTENTION!!!
		// Motorola: Big-Endien: Most Significant Bits First (Siemens)
		// Intel: Little-Endien: Least Significant Bits First (Beckhoff)
		anWriteBuffer[SIf.Cfg.uiByteOffset_wr_iOff		+0]	:= INT_TO_BYTE(SHR( THIS^.iOff,		1*8));
		anWriteBuffer[SIf.Cfg.uiByteOffset_wr_iOff		+1]	:= INT_TO_BYTE(SHR( THIS^.iOff,		0*8));
		anWriteBuffer[SIf.Cfg.uiByteOffset_wr_iBeltOn	+0]	:= INT_TO_BYTE(SHR( THIS^.iBeltOn,	1*8));
		anWriteBuffer[SIf.Cfg.uiByteOffset_wr_iBeltOn	+1]	:= INT_TO_BYTE(SHR( THIS^.iBeltOn,	0*8));
		anWriteBuffer[SIf.Cfg.uiByteOffset_wr_iManual	+0]	:= INT_TO_BYTE(SHR( THIS^.iManual,	1*8));
		anWriteBuffer[SIf.Cfg.uiByteOffset_wr_iManual	+1]	:= INT_TO_BYTE(SHR( THIS^.iManual,	0*8));
		anWriteBuffer[SIf.Cfg.uiByteOffset_wr_iRun		+0]	:= INT_TO_BYTE(SHR( THIS^.iRun,		1*8));
		anWriteBuffer[SIf.Cfg.uiByteOffset_wr_iRun		+1]	:= INT_TO_BYTE(SHR( THIS^.iRun,		0*8));
		anWriteBuffer[SIf.Cfg.uiByteOffset_wr_iSetParam	+0]	:= INT_TO_BYTE(SHR( THIS^.iSetParam,	1*8));
		anWriteBuffer[SIf.Cfg.uiByteOffset_wr_iSetParam	+1]	:= INT_TO_BYTE(SHR( THIS^.iSetParam,	0*8));
		anWriteBuffer[SIf.Cfg.uiByteOffset_wr_iGetParam	+0]	:= INT_TO_BYTE(SHR( THIS^.iGetParam,	1*8));
		anWriteBuffer[SIf.Cfg.uiByteOffset_wr_iGetParam	+1]	:= INT_TO_BYTE(SHR( THIS^.iGetParam,	0*8));
		anWriteBuffer[SIf.Cfg.uiByteOffset_wr_iAckError	+0]	:= INT_TO_BYTE(SHR( THIS^.iAckError,	1*8));
		anWriteBuffer[SIf.Cfg.uiByteOffset_wr_iAckError	+1]	:= INT_TO_BYTE(SHR( THIS^.iAckError,	0*8));
		FOR uiIdx:=0 TO SIf.Cfg.uiNumberOfModules-1 BY 1 DO
			anWriteBuffer[SIf.Cfg.uiByteOffset_wr_adiTemp_mc+0 + uiIdx*4] := DINT_TO_BYTE(SHR( THIS^.adiTemp_dc[uiIdx], 3*8));
			anWriteBuffer[SIf.Cfg.uiByteOffset_wr_adiTemp_mc+1 + uiIdx*4] := DINT_TO_BYTE(SHR( THIS^.adiTemp_dc[uiIdx], 2*8));
			anWriteBuffer[SIf.Cfg.uiByteOffset_wr_adiTemp_mc+2 + uiIdx*4] := DINT_TO_BYTE(SHR( THIS^.adiTemp_dc[uiIdx], 1*8));
			anWriteBuffer[SIf.Cfg.uiByteOffset_wr_adiTemp_mc+3 + uiIdx*4] := DINT_TO_BYTE(SHR( THIS^.adiTemp_dc[uiIdx], 0*8));
		END_FOR
		FOR uiIdx:=0 TO SIf.Cfg.uiNumberOfModules-1 BY 1 DO
			anWriteBuffer[SIf.Cfg.uiByteOffset_wr_adiAir_p+0 + uiIdx*4] := DINT_TO_BYTE(SHR( THIS^.adiAir_p[uiIdx], 3*8));
			anWriteBuffer[SIf.Cfg.uiByteOffset_wr_adiAir_p+1 + uiIdx*4] := DINT_TO_BYTE(SHR( THIS^.adiAir_p[uiIdx], 2*8));
			anWriteBuffer[SIf.Cfg.uiByteOffset_wr_adiAir_p+2 + uiIdx*4] := DINT_TO_BYTE(SHR( THIS^.adiAir_p[uiIdx], 1*8));
			anWriteBuffer[SIf.Cfg.uiByteOffset_wr_adiAir_p+3 + uiIdx*4] := DINT_TO_BYTE(SHR( THIS^.adiAir_p[uiIdx], 0*8));
		END_FOR
		anWriteBuffer[SIf.Cfg.uiByteOffset_wr_diSpeed_mm_min+0] := DINT_TO_BYTE(SHR( THIS^.diSpeed_mm_min, 3*8));
		anWriteBuffer[SIf.Cfg.uiByteOffset_wr_diSpeed_mm_min+1] := DINT_TO_BYTE(SHR( THIS^.diSpeed_mm_min, 2*8));
		anWriteBuffer[SIf.Cfg.uiByteOffset_wr_diSpeed_mm_min+2] := DINT_TO_BYTE(SHR( THIS^.diSpeed_mm_min, 1*8));
		anWriteBuffer[SIf.Cfg.uiByteOffset_wr_diSpeed_mm_min+3] := DINT_TO_BYTE(SHR( THIS^.diSpeed_mm_min, 0*8));
		
		bRememberIncrementSetParam := bIncrementSetParam;
		bIncrementSetParam := FALSE;
	END_IF

	
// Cyclic action
//--------------------------------------------------------------------------------------	
	
	// Simulation
	IF (CIf.SwCfg.bolSimulation) THEN
		me.SubStateMachine.intState := IBH_CmdState.cSTA_SUB_5;
		me.SubStateMachine.intStateNext := IBH_CmdState.cSTA_SUB_5;
	END_IF
		
	CASE me.SubStateMachine.intState OF
		
		// 1
		IBH_CmdState.cSTA_SUB_1:
			
			// Write data
			fbWrite(hLink := hLink, bExecute := FALSE );
			fbWrite(hLink := hLink,
					devAddr := SIf.Cfg.nDeviceAddress, (* Device address, MPI address of the remote component or its PROFIBUS address *)
					eArea:= eNLinkArea_DB, (* PLC data area *)
					nDB:= SIf.Cfg.nDatablockNumber, (* Data block number to which the data is written (DB, DX only) *)
					nOffset:= SIf.Cfg.nWriteStartAddress, (* Start byte/word address to which the data is send *)
					cbBuffer:= SIZEOF(anWriteBuffer), (* Contains the number of source bytes to be send *)
					pBuffer:= ADR(anWriteBuffer), (* Contains the address of the source buffer containing the data to be send *)
					bExecute:= TRUE); (* Rising edge at this input starts command execution *)
					
			me.SubStateMachine.intStateNext := IBH_CmdState.cSTA_SUB_2;
			
		// Wait and send 
		IBH_CmdState.cSTA_SUB_2:
			// check status of fbWrite
			fbWrite(hLink := hLink, bExecute := FALSE, bBusy=>bBusy, bError=>bError, nErrID=>udiErrID);
			
			// State Change Condition
			IF NOT bBusy THEN
				Out_udiDriverErrorID := udiErrID;
				IF bError THEN
					Out_bDriverError := TRUE;
					me.StateMachine.intStateNext := IBH_CmdState.cSTA_DISCONNECTBusy;
				ELSE
					Out_bDriverError := FALSE;
					IF bRememberIncrementSetParam THEN
						me.SubStateMachine.intStateNext := IBH_CmdState.cSTA_SUB_3;
					ELSE
						me.SubStateMachine.intStateNext := IBH_CmdState.cSTA_SUB_5;
					END_IF
				END_IF
			END_IF
			
		// 3
		IBH_CmdState.cSTA_SUB_3:
			bRememberIncrementSetParam := FALSE;
			IF (iSetParam = MAX_INT OR iSetParam < 0) THEN
				iSetParam := 0;
			END_IF
			iSetParam := iSetParam + 1;
		
			// Adapt Write Buffer
			anWriteBuffer[SIf.Cfg.uiByteOffset_wr_iSetParam	+0]	:= INT_TO_BYTE(SHR( THIS^.iSetParam,	1*8));
			anWriteBuffer[SIf.Cfg.uiByteOffset_wr_iSetParam	+1]	:= INT_TO_BYTE(SHR( THIS^.iSetParam,	0*8));
			
			// Write data
			fbWrite(hLink := hLink, bExecute := FALSE );
			fbWrite(hLink := hLink,
					devAddr := SIf.Cfg.nDeviceAddress, (* Device address, MPI address of the remote component or its PROFIBUS address *)
					eArea:= eNLinkArea_DB, (* PLC data area *)
					nDB:= SIf.Cfg.nDatablockNumber, (* Data block number to which the data is written (DB, DX only) *)
					nOffset:= SIf.Cfg.nWriteStartAddress, (* Start byte/word address to which the data is send *)
					cbBuffer:= SIZEOF(anWriteBuffer), (* Contains the number of source bytes to be send *)
					pBuffer:= ADR(anWriteBuffer), (* Contains the address of the source buffer containing the data to be send *)
					bExecute:= TRUE); (* Rising edge at this input starts command execution *)
			
			me.SubStateMachine.intStateNext := IBH_CmdState.cSTA_SUB_4;
			
		// 4
		IBH_CmdState.cSTA_SUB_4:
			
			// check status of fbWrite
			fbWrite(hLink := hLink, bExecute := FALSE, bBusy=>bBusy, bError=>bError, nErrID=>udiErrID);
			
			// State Change Condition
			IF NOT bBusy THEN
				Out_udiDriverErrorID := udiErrID;
				IF bError THEN
					Out_bDriverError := TRUE;
					me.StateMachine.intStateNext := IBH_CmdState.cSTA_DISCONNECTBusy;
				ELSE
					Out_bDriverError := FALSE;
					me.SubStateMachine.intStateNext := IBH_CmdState.cSTA_SUB_5;
				END_IF
			END_IF
			
		// 5
		IBH_CmdState.cSTA_SUB_5:
			me.StateMachine.intStateNext := IBH_CmdState.cSTA_WRITE;
			
	END_CASE
		

// Exit action
//--------------------------------------------------------------------------------------
	IF (me.StateMachine.intState <> me.StateMachine.intStateNext) THEN
		// state is going to change
		;
	END_IF
                      
END_METHOD

{attribute 'object_name' := 'sta_WRITE'}
METHOD sta_WRITE : BOOL
                        // state implemetation

// Entry action
//--------------------------------------------------------------------------------------
	IF (me.StateMachine.intState <> me.StateMachine.intStateLastCycle) THEN
		// state changed since last cycle
		me.StateMachine.intStateLastCycle := me.StateMachine.intState;
	END_IF

	
// Cyclic action
//--------------------------------------------------------------------------------------	
	// Simulation
	IF (CIf.SwCfg.bolSimulation) THEN
		;
	END_IF
	
	// State Change Condition
	CASE me.intCmd OF
		// OFF
		Base_PLC.cCMD_OFF:
			me.StateMachine.intStateNext := IBH_CmdState.cSTA_DISCONNECTBusy;
	ELSE
		// DEFAULT
		me.StateMachine.intStateNext := IBH_CmdState.cSTA_READBusy;
	END_CASE


// Exit action
//--------------------------------------------------------------------------------------
	IF (me.StateMachine.intState <> me.StateMachine.intStateNext) THEN
		// state is going to change
		;
	END_IF
                      
END_METHOD

{attribute 'object_name' := 'sta_DISCONNECT'}
METHOD sta_DISCONNECT : BOOL
                        // state implemetation

// Entry action
//--------------------------------------------------------------------------------------
	IF (me.StateMachine.intState <> me.StateMachine.intStateLastCycle) THEN
		// state changed since last cycle
		me.StateMachine.intStateLastCycle := me.StateMachine.intState;
	END_IF

	
// Cyclic action
//--------------------------------------------------------------------------------------	
	// Simulation
	IF (CIf.SwCfg.bolSimulation) THEN
		;
	END_IF
	
	// State Change Condition
	CASE me.intCmd OF
		// OFF
		Base_PLC.cCMD_OFF:
			me.StateMachine.intStateNext := BASE_PLC.cSTA_OFFBusy;
	ELSE
		// DEFAULT
		me.StateMachine.intStateNext := IBH_CmdState.cSTA_CONNECTBusy;
	END_CASE


// Exit action
//--------------------------------------------------------------------------------------
	IF (me.StateMachine.intState <> me.StateMachine.intStateNext) THEN
		// state is going to change
		;
	END_IF
                      
END_METHOD

{attribute 'object_name' := 'getCtrlSIf'}
METHOD getCtrlSIf : POINTER TO T_Ctrl_SIf_IBH
                        getCtrlSIf := ADR(SIf);
                      
END_METHOD

{attribute 'object_name' := 'sta_READ'}
METHOD sta_READ : BOOL
  VAR
    uiIdx : UINT;
  END_VAR
                        // state implemetation

// Entry action
//--------------------------------------------------------------------------------------
	IF (me.StateMachine.intState <> me.StateMachine.intStateLastCycle) THEN
		me.StateMachine.intStateLastCycle := me.StateMachine.intState;
	END_IF

	
// Cyclic action
//--------------------------------------------------------------------------------------	
	
	// Simulation
	IF (CIf.SwCfg.bolSimulation) THEN
		THIS^.Out_iStatus	:= iSimStatus;
		THIS^.Out_bOff		:= bSimOff;
		THIS^.Out_bBeltOn	:= bSimBeltOn;
		THIS^.Out_bManual	:= bSimManual;
		THIS^.Out_bRun		:= bSimRun;
		THIS^.Out_bSetParam	:= FALSE;
		THIS^.Out_bGetParam	:= FALSE;
		THIS^.Out_bAckError	:= FALSE;
		
		IF bSimRun THEN
			Out_adiTemp_dc := adiTemp_dc;
			Out_adiAir_p := adiAir_p;
		ELSE
			FOR uiIdx:=0 TO SIf.Cfg.uiNumberOfModules BY 1 DO
				THIS^.Out_adiTemp_dc[uiIdx] := 0;
				THIS^.Out_adiAir_p[uiIdx] := 0;
			END_FOR
		END_IF
		
		IF bSimRun OR bSimBeltOn THEN
			Out_diSpeed_mm_min := diSpeed_mm_min;
		ELSE
			THIS^.Out_diSpeed_mm_min :=	0;
		END_IF
		
		THIS^.Out_iErrorLevel := 0;
		THIS^.Out_iErrorID := 0;
	ELSE
		// Analyse Read Buffer
		// !!!ATTENTION!!!
		// Motorola: Big-Endien: Most Significant Bits First (Siemens)
		// Intel: Little-Endien: Least Significant Bits First (Beckhoff)
		THIS^.Out_iStatus :=		SHL(BYTE_TO_INT(anReadBuffer[SIf.Cfg.uiByteOffset_rd_iStatus+0]),1*8)
								+	SHL(BYTE_TO_INT(anReadBuffer[SIf.Cfg.uiByteOffset_rd_iStatus+1]),0*8);
		THIS^.Out_bOff		:= bitAccess( anReadBuffer[SIf.Cfg.uiByteOffset_rd_bOff]		,SIf.Cfg.uiBitOffset_rd_bOff);
		THIS^.Out_bBeltOn	:= bitAccess( anReadBuffer[SIf.Cfg.uiByteOffset_rd_bBeltOn]		,SIf.Cfg.uiBitOffset_rd_bBeltOn);
		THIS^.Out_bManual	:= bitAccess( anReadBuffer[SIf.Cfg.uiByteOffset_rd_bManual]		,SIf.Cfg.uiBitOffset_rd_bManual);
		THIS^.Out_bRun		:= bitAccess( anReadBuffer[SIf.Cfg.uiByteOffset_rd_bRun]		,SIf.Cfg.uiBitOffset_rd_bRun);
		THIS^.Out_bSetParam	:= bitAccess( anReadBuffer[SIf.Cfg.uiByteOffset_rd_bSetParam]	,SIf.Cfg.uiBitOffset_rd_bSetParam);
		THIS^.Out_bGetParam	:= bitAccess( anReadBuffer[SIf.Cfg.uiByteOffset_rd_bGetParam]	,SIf.Cfg.uiBitOffset_rd_bGetParam);
		THIS^.Out_bAckError	:= bitAccess( anReadBuffer[SIf.Cfg.uiByteOffset_rd_bAckError]	,SIf.Cfg.uiBitOffset_rd_bAckError);
		FOR uiIdx:=0 TO SIf.Cfg.uiNumberOfModules BY 1 DO
			THIS^.Out_adiTemp_dc[uiIdx] :=		SHL(BYTE_TO_DINT(anReadBuffer[SIf.Cfg.uiByteOffset_rd_adiTemp_mc+0 + uiIdx*4]),3*8)
											+	SHL(BYTE_TO_DINT(anReadBuffer[SIf.Cfg.uiByteOffset_rd_adiTemp_mc+1 + uiIdx*4]),2*8)
											+	SHL(BYTE_TO_DINT(anReadBuffer[SIf.Cfg.uiByteOffset_rd_adiTemp_mc+2 + uiIdx*4]),1*8)
											+	SHL(BYTE_TO_DINT(anReadBuffer[SIf.Cfg.uiByteOffset_rd_adiTemp_mc+3 + uiIdx*4]),0*8);
		END_FOR
		FOR uiIdx:=0 TO SIf.Cfg.uiNumberOfModules BY 1 DO
			THIS^.Out_adiAir_p[uiIdx] :=		SHL(BYTE_TO_DINT(anReadBuffer[SIf.Cfg.uiByteOffset_rd_adiAir_p+0 + uiIdx*4]),3*8)
											+	SHL(BYTE_TO_DINT(anReadBuffer[SIf.Cfg.uiByteOffset_rd_adiAir_p+1 + uiIdx*4]),2*8)
											+	SHL(BYTE_TO_DINT(anReadBuffer[SIf.Cfg.uiByteOffset_rd_adiAir_p+2 + uiIdx*4]),1*8)
											+	SHL(BYTE_TO_DINT(anReadBuffer[SIf.Cfg.uiByteOffset_rd_adiAir_p+3 + uiIdx*4]),0*8);
		END_FOR
		THIS^.Out_diSpeed_mm_min :=		SHL(BYTE_TO_DINT(anReadBuffer[SIf.Cfg.uiByteOffset_rd_diSpeed_mm_min+0]),3*8)
									+	SHL(BYTE_TO_DINT(anReadBuffer[SIf.Cfg.uiByteOffset_rd_diSpeed_mm_min+1]),2*8)
									+	SHL(BYTE_TO_DINT(anReadBuffer[SIf.Cfg.uiByteOffset_rd_diSpeed_mm_min+2]),1*8)
									+	SHL(BYTE_TO_DINT(anReadBuffer[SIf.Cfg.uiByteOffset_rd_diSpeed_mm_min+3]),0*8);
		THIS^.Out_iErrorLevel :=		SHL(BYTE_TO_INT(anReadBuffer[SIf.Cfg.uiByteOffset_rd_iErrorLevel+0]),1*8)
									+	SHL(BYTE_TO_INT(anReadBuffer[SIf.Cfg.uiByteOffset_rd_iErrorLevel+1]),0*8);
		THIS^.Out_iErrorID :=			SHL(BYTE_TO_INT(anReadBuffer[SIf.Cfg.uiByteOffset_rd_iErrorID+0]),1*8)
									+	SHL(BYTE_TO_INT(anReadBuffer[SIf.Cfg.uiByteOffset_rd_iErrorID+1]),0*8);
	END_IF
									
	// State Change Condition
	CASE me.intCmd OF
		// OFF
		Base_PLC.cCMD_OFF:
			me.StateMachine.intStateNext := IBH_CmdState.cSTA_DISCONNECTBusy;
	ELSE
		// DEFAULT
		me.StateMachine.intStateNext := IBH_CmdState.cSTA_WRITEBusy;
	END_CASE


// Exit action
//--------------------------------------------------------------------------------------
	IF (me.StateMachine.intState <> me.StateMachine.intStateNext) THEN
		// state is going to change
		;
	END_IF
                      
END_METHOD

{attribute 'object_name' := 'sta_PONBusy'}
METHOD sta_PONBusy : BOOL
                        // state implemetation

// Entry action
//--------------------------------------------------------------------------------------
	IF (me.StateMachine.intState <> me.StateMachine.intStateLastCycle) THEN
		// state changed since last cycle
		me.StateMachine.intStateLastCycle := me.StateMachine.intState;
	END_IF

	
// Cyclic action
//--------------------------------------------------------------------------------------	
	// Simulation
	IF (CIf.SwCfg.bolSimulation) THEN
		;
	END_IF

	// State Change Condition
	me.StateMachine.intStateNext := Base_PLC.cSTA_PON;


// Exit action
//--------------------------------------------------------------------------------------
	IF (me.StateMachine.intState <> me.StateMachine.intStateNext) THEN
		// state is going to change
		;
	END_IF
                      
END_METHOD

{attribute 'object_name' := 'sta_OFFBusy'}
METHOD sta_OFFBusy : BOOL
                        // state implemetation

// Entry action
//--------------------------------------------------------------------------------------
	IF (me.StateMachine.intState <> me.StateMachine.intStateLastCycle) THEN
		// state changed since last cycle
		me.StateMachine.intStateLastCycle := me.StateMachine.intState;
	END_IF

	
// Cyclic action
//--------------------------------------------------------------------------------------	
	// Simulation
	IF (CIf.SwCfg.bolSimulation) THEN
		;
	END_IF
	
	// Reset Output
	Out_bDriverError := FALSE;
	Out_udiDriverErrorID := 0;
	
	// State Change Condition
	me.StateMachine.intStateNext := Base_PLC.cCMD_OFF;


// Exit action
//--------------------------------------------------------------------------------------
	IF (me.StateMachine.intState <> me.StateMachine.intStateNext) THEN
		// state is going to change
		;
	END_IF
                      
END_METHOD

{attribute 'object_name' := 'StateMachine'}
METHOD StateMachine : BOOL
                        SUPER^.StateMachine();

// main statemachine of base controller
CASE me.StateMachine.intState OF
	// CONNECT
    IBH_CmdState.cSTA_CONNECT: 
        THIS^.sta_CONNECT();
    IBH_CmdState.cSTA_CONNECTBusy: 
        THIS^.sta_CONNECTBusy();
	// WRITE
	IBH_CmdState.cSTA_WRITE: 
        THIS^.sta_WRITE();
    IBH_CmdState.cSTA_WRITEBusy: 
        THIS^.sta_WRITEBusy();
	// READ
	IBH_CmdState.cSTA_READ: 
        THIS^.sta_READ();
    IBH_CmdState.cSTA_READBusy: 
        THIS^.sta_READBusy();
	// DISCONNECT
	IBH_CmdState.cSTA_DISCONNECT: 
        THIS^.sta_DISCONNECT();
    IBH_CmdState.cSTA_DISCONNECTBusy: 
        THIS^.sta_DISCONNECTBusy();
END_CASE;
                      
END_METHOD

{attribute 'object_name' := 'getCmdState'}
METHOD getCmdState : STRING
  VAR_INPUT
    intCmdState : INT;
    bolState : BOOL;
  END_VAR
                        getCmdState := SUPER^.getCmdState(intCmdState:=intCmdState,bolState:=bolState); // get global/base defined cmds/states

IF (getCmdState='') THEN // global not defined get local
	// get string cmd/state string information in runtime
	IF (bolState=FALSE) THEN
		// cmd's
		CASE intCmdState OF
			IBH_CmdState.cCMD_CONNECT:
				getCmdState := 'CONNECT';
			IBH_CmdState.cCMD_WRITE:
				getCmdState := 'WRITE';
			IBH_CmdState.cCMD_READ:
				getCmdState := 'READ';
			IBH_CmdState.cCMD_DISCONNECT:
				getCmdState := 'DISCONNECT';
		ELSE
			getCmdState := 'Cmd not defined';
		END_CASE;
	ELSE
		// state's
		CASE intCmdState OF
			// CONNECT
			IBH_CmdState.cSTA_CONNECTBusy: 
				getCmdState := 'CONNECTBusy';
			IBH_CmdState.cSTA_CONNECT: 
				getCmdState := 'CONNECT';
			// WRITE
			IBH_CmdState.cSTA_WRITEBusy: 
				getCmdState := 'WRITEBusy';
			IBH_CmdState.cSTA_WRITE: 
				getCmdState := 'WRITE';
			// READ
			IBH_CmdState.cSTA_READBusy: 
				getCmdState := 'READBusy';
			IBH_CmdState.cSTA_READ: 
				getCmdState := 'READ';
			// DISCONNECT
			IBH_CmdState.cSTA_DISCONNECTBusy: 
				getCmdState := 'DISCONNECTBusy';
			IBH_CmdState.cSTA_DISCONNECT: 
				getCmdState := 'DISCONNECT';
		ELSE
			getCmdState := 'State not defined';
		END_CASE
	END_IF
END_IF
                      
END_METHOD

{attribute 'object_name' := 'setAirflow'}
METHOD setAirflow
  VAR_INPUT
    In_adiAir_p : ARRAY[1..MAX_NUMBER_OF_OVEN_MODULES] OF DINT;  (* Airflow in % *)
  END_VAR
                        adiAir_p := In_adiAir_p;
bIncrementSetParam := TRUE;
                      
END_METHOD

{attribute 'object_name' := 'Always'}
METHOD Always : BOOL
  VAR
    fbOVN : INT;
  END_VAR
                        // ----------------------------------------------------------------------------------
// Conditions Always
IF (me.bolChangeBackToAUTO=TRUE) THEN // switch mode to automatic switch off controller
	me.StateMachine.intStateNext := cSTA_OFFBusy;
	me.bolChangeBackToAUTO := FALSE;
END_IF

IF (CIf.SwCfg.bolExist=FALSE) THEN // hardware of controller does not exist
	me.StateMachine.intStateNext := cSTA_SINGLE_ANSWER;
ELSE
	IF (((me.StateMachine.intState=cSTA_INITIALIZED) OR (me.intCmd=cCMD_PON)) 
		AND (me.StateMachine.intState<>cSTA_PONBusy) AND (me.StateMachine.intState<>cSTA_PON)
		AND (me.StateMachine.intState<>cSTA_ERROR) AND (me.StateMachine.intState<>cSTA_ERRORQuit) 
		AND (me.StateMachine.intState<>cSTA_EOFF) AND (me.StateMachine.intState<>cSTA_EOFFBusy)) THEN // switch after startup to PONBusy
		me.StateMachine.intStateNext := cSTA_PONBusy;
		
	ELSIF (((me.Alarm.eActivAlmClass=E_AlmClass.EOFF) OR (me.intCmd=cCMD_EOFF)) 
		AND (me.StateMachine.intState<>cSTA_ERROR) AND (me.StateMachine.intState<>cSTA_ERRORQuit) 
		AND (me.StateMachine.intState<>cSTA_EOFF) AND (me.StateMachine.intState<>cSTA_EOFFBusy)
		AND (me.StateMachine.intState>cSTA_PON)) THEN
		me.StateMachine.intStateNext := cSTA_EOFFBusy;
	
	ELSIF (((me.Alarm.eActivAlmClass=E_AlmClass.OFF) (*OR (me.intCmd=cCMD_OFF)*))
		AND (me.StateMachine.intState<>cSTA_ERROR) AND (me.StateMachine.intState<>cSTA_ERRORQuit)
		AND (me.StateMachine.intState<>cSTA_EOFF) AND (me.StateMachine.intState<>cSTA_EOFFBusy)
		AND (me.StateMachine.intState<>cSTA_OFF) AND (me.StateMachine.intState<>cSTA_OFFBusy)
		AND (me.StateMachine.intState>cSTA_PON)) THEN
		me.StateMachine.intStateNext := cSTA_OFFBusy;
	
	END_IF
	
	IF		NOT CIf.SwCfg.bolEnable
		AND (me.StateMachine.intState<>cSTA_OFF)
		AND (me.StateMachine.intState<>cSTA_OFFBusy) THEN
		CIf.Job.intACmd := cCMD_OFF;
	END_IF
	
	Out_bDriverConnected := FALSE;
	IF		(me.StateMachine.intState=cSTA_WRITE) OR (me.StateMachine.intState=cSTA_WRITEBusy)
		OR	(me.StateMachine.intState=cSTA_READ) OR (me.StateMachine.intState=cSTA_READBusy) THEN
		Out_bDriverConnected := TRUE;
	END_IF
	
END_IF

// ----------------------------------------------------------------------------------
// overrule error always from base -> no EOFF State!! in EOFF go to OFF
IF (me.StateMachine.intStateNext = cSTA_EOFFBusy) THEN
	IF (me.StateMachine.intState = cSTA_OFF) THEN
		me.StateMachine.intStateNext := cSTA_OFF;
	ELSE // stay in OFF
		me.StateMachine.intStateNext := cSTA_OFFBusy;
	END_IF
END_IF
                      
END_METHOD

{attribute 'object_name' := 'setSpeed'}
METHOD setSpeed
  VAR_INPUT
    In_diSpeed_mm_min : DINT;  (* Belt speed in mm/min *)
  END_VAR
                        diSpeed_mm_min := In_diSpeed_mm_min;
bIncrementSetParam := TRUE;
                      
END_METHOD

{attribute 'object_name' := 'sta_CONNECT'}
METHOD sta_CONNECT : BOOL
                        // state implemetation

// Entry action
//--------------------------------------------------------------------------------------
	IF (me.StateMachine.intState <> me.StateMachine.intStateLastCycle) THEN
		// state changed since last cycle
		me.StateMachine.intStateLastCycle := me.StateMachine.intState;
	END_IF

	
// Cyclic action
//--------------------------------------------------------------------------------------	
	// Simulation
	IF (CIf.SwCfg.bolSimulation) THEN
		;
	END_IF
	
	// State Change Condition
	CASE me.intCmd OF
		// OFF
		Base_PLC.cCMD_OFF:
			me.StateMachine.intStateNext := IBH_CmdState.cSTA_DISCONNECTBusy;
	ELSE
		// DEFAULT
		me.StateMachine.intStateNext := IBH_CmdState.cSTA_WRITEBusy;
	END_CASE


// Exit action
//--------------------------------------------------------------------------------------
	IF (me.StateMachine.intState <> me.StateMachine.intStateNext) THEN
		// state is going to change
		;
	END_IF
                      
END_METHOD

{attribute 'object_name' := 'sta_DISCONNECTBusy'}
METHOD sta_DISCONNECTBusy : BOOL
  VAR
    bBusy : BOOL;
    bError : BOOL;
    udiErrID : UDINT;
  END_VAR
                        // state implemetation

// Entry action
//--------------------------------------------------------------------------------------
	IF (me.StateMachine.intState <> me.StateMachine.intStateLastCycle) THEN
		// state changed since last cycle
		me.StateMachine.intStateLastCycle := me.StateMachine.intState;
		
		IF NOT CIf.SwCfg.bolSimulation THEN
			// Close connection
			fbClose(hLink := hLink, bExecute := FALSE);
			fbClose(hLink := hLink, bExecute := TRUE);
		END_IF
	END_IF

	
// Cyclic action
//--------------------------------------------------------------------------------------	
	
	// check status of fbClose
	fbClose(hLink := hLink, bExecute := FALSE, bBusy=>bBusy, bError=>bError, nErrID=>udiErrID);
	
	// Simulation
	IF (CIf.SwCfg.bolSimulation) THEN
		bBusy := FALSE;
		bError := FALSE;
		udiErrID := 0;
	END_IF
	
	// State Change Condition
	IF NOT bBusy THEN
		Out_udiDriverErrorID := udiErrID;
		IF bError THEN
			Out_bDriverError := TRUE;
		ELSE
			Out_bDriverError := FALSE;
		END_IF
		me.StateMachine.intStateNext := IBH_CmdState.cSTA_DISCONNECT;
	END_IF

// Exit action
//--------------------------------------------------------------------------------------
	IF (me.StateMachine.intState <> me.StateMachine.intStateNext) THEN
		// state is going to change
		;
	END_IF
                      
END_METHOD

PROPERTY CtrlSIf : POINTER TO T_Ctrl_SIf_IBH
GET
                          CtrlSIf := ADR(SIf);
                        
END_GET
END_PROPERTY
END_FUNCTION_BLOCK

FUNCTION_BLOCK FB_POD
  VAR_INPUT
    In_bolHomeSwitch : BOOL;  (* home switch - only active if configured *)
  END_VAR
  VAR
    bolInitDone : BOOL;
    bolActivate : BOOL := TRUE;
    SIf : T_POD;  (* driver specific interface *)
    stAxisParameter : ST_AxisParameterSet;  (* complete parameter set of the axis *)
    fbAxis : AXIS_REF;  (* axis reference (process data plc/nc) *)
    stStateMachine : T_POD_StateMachine;  (* /// get direct drive state of yaskawa /// access over mapping!! {attribute 'TcLinkTo':='TIID^Device 1 (EtherCAT)^Box 1 (SGDV-E1 CoE Drive)^2nd Transmit PDO mapping^Status word'} In_worPOD_DriveState AT %I*: WORD; /// get direct drive inputs of yaskawa /// access over mapping!! {attribute 'TcLinkTo':='TIID^Device 1 (EtherCAT)^Box 1 (SGDV-E1 CoE Drive)^2nd Transmit PDO mapping^Status word'} In_udiPOD_DriveInputs AT %I*: UDINT; *)
    usiCase : USINT;  (* case variable *)
    usiCaseScmd : USINT;  (* case variable for service cmd's *)
    fbMcPower : MC_Power;  (* PlcOpen standard FUB's enable and override *)
    fbMcReset : MC_Reset;
    fbMcHalt : MC_Halt;
    fbMcAbsMove : MC_MoveAbsolute;
    fbMcModMove : MC_MoveModulo;
    fbMcRelMove : MC_MoveRelative;
    fbMcMoveVelocity : MC_MoveVelocity;
    fbMcJog : MC_Jog;
    fbMCStop : MC_Stop;
    fbMcHome : MC_Home;
    fbMCReadParameterSet : MC_ReadParameterSet;  (* The complete parameter set of an axis can be read with the function block MC_ReadParameterSet. *)
    fbMCReadDriveAdress : MC_ReadDriveAddress;  (* MC_ReadDriveAddress reads the ADS information that is required to access a drive device connected to an axis. *)
    fbMCWriteParameter : MC_WriteParameter;
    fbMCWriteBoolParameter : MC_WriteBoolParameter;
    fbMCReadParameter : MC_ReadParameter;
    fbMCReadBoolParameter : MC_ReadBoolParameter;
    fbMCReadAxisError : MC_ReadAxisError;
    fbEcCoeSdoWrite : FB_EcCoeSdoWrite;  (* Ethercat standard FUB' *)
    fbEcCoeSdoRead : FB_EcCoeSdoRead;
    fbEcSetSlaveState : FB_EcSetSlaveState;  (* set ethercat mode preop/op *)
    sinValue : SINT;  (* help values for parameter handling *)
    intValue : INT;
    dinValue : DINT;
    usiValue : USINT;
    uinValue : UINT;
    udiValue : UDINT;
    bolfpFirstCycleDone : BOOL;  (* help value for FUB handling *)
    fbSimTON : TC2_STANDARD.TON;
    udiSimPosTime_ms : UDINT;
    lreSimJogSpeed : LREAL;
    lreActPos_old : LREAL;
  END_VAR

                  (*__________________________________________________________________________________________________
¦	
¦	Vistaprint Schweiz GmbH
¦	CH - 8401 Winterthur
¦
¦	www.vistaprint.ch - info@vistaprint.ch
¦___________________________________________________________________________________________________

Function desription:
PLC open driver for servo drives.


History:
Version		Date			Author		Comment
---------------------------------------------------------------------------------------------------
0.00.1		18.06.2013		AVME/KVO	Start history
0.00.2		22.09.2014		AVME/MRU	Rework for Beckhoff Servo Drives
0.00.3		12.12.2014		AVME/MRU	Add cCMD_OFF
___________________________________________________________________________________________________*)


IF (bolActivate) THEN // cyclic call enabled
	
	IF (bolInitDone=FALSE) THEN // first cycle -> init
		CtrlInit();
		bolInitDone := TRUE;
	ELSE
		CycleStartDuty();
		
		StateMachine_Service(); // handles asynchron service commands
		
		StateMachine();
		
		CycleEndDuty();
	END_IF
	
END_IF;
                

{attribute 'object_name' := 'sta_PowerOnBusy'}
METHOD sta_PowerOnBusy : BOOL
                        // state implemetation
//--------------------------------------------------------------------------------------
// Entry action
	IF (stStateMachine.intState<>stStateMachine.intStateLastCycle) THEN
		stStateMachine.intStateLastCycle := stStateMachine.intState;
		
	END_IF


